		IF bPackBarcode THEN
			sOutBarcode	:= sPackBarcode;
		ELSIF bOuterBarcode THEN
			sOutBarcode := F_CODE_GetItem(sOuterBarcode, eCodeAIType.SerialCode, stCodeInfo_Outer);
		ELSIF bCaseBarcode THEN
			(*fbDecodeGS1(strGS1String := CONCAT(']d2',sCaseBarcode), bDontParseAsGS1 := TRUE, strBarcode => sOutBarcode);*)
			sOutBarcode	:= sCaseBarcode;
		ELSE
			sOutBarcode := '';
		END_IF

		bScanDone := TRUE;

	ELSIF bEnableInvalidSearch AND NOT bEnableCaseContentSearch AND NOT bEnablePackCodeRefeed THEN

		sNewPackCodeRefeed := '';

		IF bPackBarcode THEN
			sOutBarcode :=  F_CODE_GetItem(sPackBarcode, eCodeAIType.SerialCode, stCodeInfo_Pack);
		ELSIF bOuterIntermediate THEN
			sOutBarcode := F_CODE_GetItem(sOuterIntermediateBarcode, eCodeAIType.SerialCode, stCodeInfo_Intermediate);
		ELSIF bOuterBarcode THEN
			sOutBarcode := F_CODE_GetItem(sOuterBarcode, eCodeAIType.SerialCode, stCodeInfo_Outer);
		ELSE
			sOutBarcode := '';
		END_IF

		bScanDone := TRUE;

	ELSIF bEnableInvalidSearch AND NOT bEnableCaseContentSearch AND bEnablePackCodeRefeed THEN

		IF bPackBarcode THEN
			sOutBarcode := F_CODE_GetItem(sPackBarcode, eCodeAIType.SerialCode, stCodeInfo_Pack);
			sNewPackCodeRefeed := sPackBarcode;
		ELSE
			sOutBarcode := '';
			sNewPackCodeRefeed := '';
		END_IF

		bScanDone := TRUE;

	ELSE

		sOutBarcode := '';
		sNewPackCodeRefeed := '';

	END_IF

	(* set output *)
	bBusy := FALSE;
	bDone := TRUE;
END_IF

END_FUNCTION_BLOCK

// ---- POUs/METS/Common LIB/09_SYSTEM LIB/FB_SYSTEM_SeqControl.TcPOU
FUNCTION_BLOCK FB_SYSTEM_SeqControl
VAR_INPUT
	nSeqStepNo	: INT;
END_VAR
VAR_OUTPUT
	bActive		: BOOL;
	bStep00		: BOOL;
	bStep01		: BOOL;
	bStep02		: BOOL;
	bStep03		: BOOL;
	bStep04		: BOOL;
	bStep05		: BOOL;
	bStep06		: BOOL;
	bStep07		: BOOL;
	bStep08		: BOOL;
	bStep09		: BOOL;
	bStep10		: BOOL;
	bStep11		: BOOL;
	bStep12		: BOOL;
	bStep13		: BOOL;
	bStep14		: BOOL;
	bStep15		: BOOL;
	bStep16		: BOOL;
	bStep17		: BOOL;
	bStep18		: BOOL;
	bStep19		: BOOL;
	bStep20		: BOOL;
END_VAR
VAR
END_VAR
(*
-------------------------------------------------------------------------------------------------
Date		Version	Author	Comments
-------------------------------------------------------------------------------------------------
30/01/2015	3.00.00	PB		Initial release

-------------------------------------------------------------------------------------------------
*)

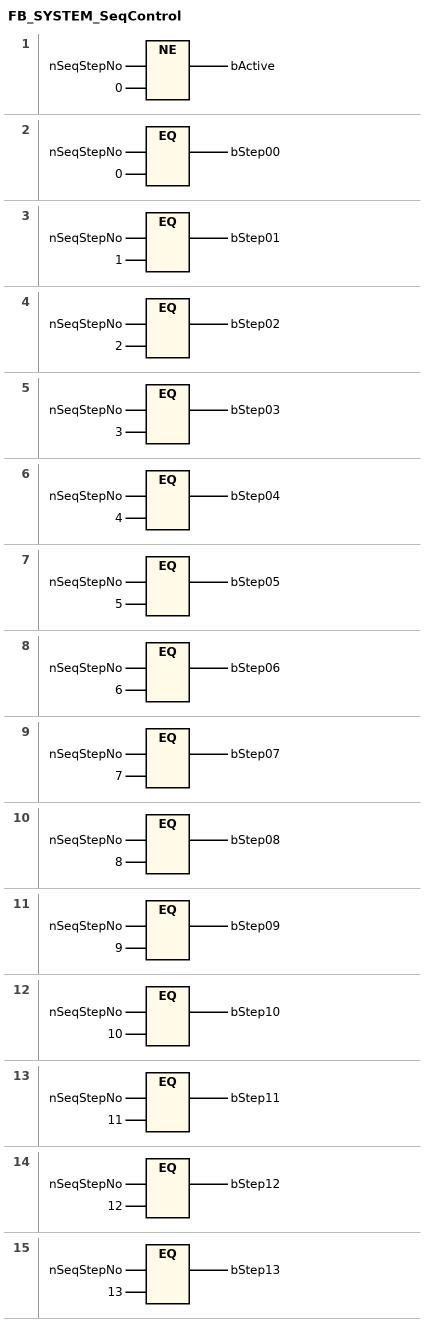
// NETWORK 1
bActive := nSeqStepNo <> 0;

// NETWORK 2
bStep00 := nSeqStepNo = 0;

// NETWORK 3
bStep01 := nSeqStepNo = 1;

// NETWORK 4
bStep02 := nSeqStepNo = 2;

// NETWORK 5
bStep03 := nSeqStepNo = 3;

// NETWORK 6
bStep04 := nSeqStepNo = 4;

// NETWORK 7
bStep05 := nSeqStepNo = 5;

// NETWORK 8
bStep06 := nSeqStepNo = 6;

// NETWORK 9
bStep07 := nSeqStepNo = 7;

// NETWORK 10
bStep08 := nSeqStepNo = 8;

// NETWORK 11
bStep09 := nSeqStepNo = 9;

// NETWORK 12
bStep10 := nSeqStepNo = 10;

// NETWORK 13
bStep11 := nSeqStepNo = 11;

// NETWORK 14
bStep12 := nSeqStepNo = 12;

// NETWORK 15
bStep13 := nSeqStepNo = 13;

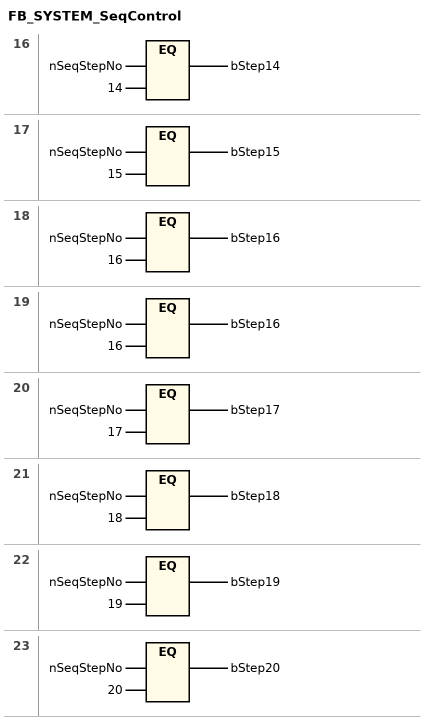
// NETWORK 16
bStep14 := nSeqStepNo = 14;

// NETWORK 17
bStep15 := nSeqStepNo = 15;

// NETWORK 18
bStep16 := nSeqStepNo = 16;

// NETWORK 19
bStep16 := nSeqStepNo = 16;

// NETWORK 20
bStep17 := nSeqStepNo = 17;

// NETWORK 21
bStep18 := nSeqStepNo = 18;

// NETWORK 22
bStep19 := nSeqStepNo = 19;

// NETWORK 23
bStep20 := nSeqStepNo = 20;

END_FUNCTION_BLOCK

// ---- POUs/METS/Common LIB/09_SYSTEM LIB/FB_SYSTEM_ShiftMonitor.TcPOU
FUNCTION_BLOCK FB_SYSTEM_ShiftMonitor
VAR_INPUT
	bEnable				: BOOL;
	stSystemTime			: TIMESTRUCT;
END_VAR
VAR_IN_OUT

	stPCMStatus				: ST_PCM_Status;	(* PCMstatus *)
	aShiftSchedule				: ARRAY[1..cSHIFTNUMBER] OF TIMESTRUCT;
	aShiftChangeActive		: ARRAY[1..cSHIFTNUMBER] OF BOOL;
	stCurrentStatisticNV		: ST_NOVRAM_METS_EventCounters;
	stCSVStoreTable			: ST_HMI_CSVStoreTable;

END_VAR
VAR_OUTPUT

	bShiftChanged				: BOOL;
	stLastShift					: TIMESTRUCT;
END_VAR
VAR
	fbExecute					: R_TRIG;
	nNumberShift				: T_PositiveINT;
	bEndOfShift				: BOOL;
	(*nActiveShiftCounter		: INT;*)

END_VAR

(* shift manager disabled *)
IF NOT bEnable  THEN

	(* clear outputs *)
	bEndOfShift := FALSE;
	MEMSET(ADR(stLastShift), 16#00, SIZEOF(stLastShift));
	RETURN;
END_IF


IF stCurrentStatisticNV.stEventStartDT.wYear = 0 AND stCurrentStatisticNV.stEventStartDT.wMonth = 0 THEN
	stCurrentStatisticNV.stEventStartDT := stSystemTime;
	stCurrentStatisticNV.nShiftID 		:= 1;
END_IF
(*
nActiveShiftCounter := 0;

FOR nNumberShift := 1 TO cSHIFTNUMBER DO

	IF	aShiftChangeActive[nNumberShift] 	THEN
		nActiveShiftCounter := nActiveShiftCounter + 1;
	END_IF
END_FOR
*)
FOR nNumberShift := 1 TO cSHIFTNUMBER DO

	IF	aShiftChangeActive[nNumberShift] 							AND
		aShiftSchedule[nNumberShift].wHour  = stSystemTime.wHour 		AND
		aShiftSchedule[nNumberShift].wMinute = stSystemTime.wMinute 	(*AND
		aShiftSchedule[nNumberShift].wSecond = .sSystemTime.wSecond*)		THEN

		(*stCurrentStatisticNV.stEventEndDT	:= stSystemTime;*)
		bEndOfShift := TRUE;
		EXIT;
	ELSE
		bEndOfShift := FALSE;
	END_IF
END_FOR

(*
IF nActiveShiftCounter <> 0 THEN
	stCurrentStatisticNV.stEndShiftDT := F_ApplyTimeOffset(stCurrentStatisticNV.stStartShiftDT, 86400000/nActiveShiftCounter);
ELSE
	stCurrentStatisticNV.stEndShiftDT := F_ApplyTimeOffset(stCurrentStatisticNV.stStartShiftDT, 86400000);
END_IF
*)
(***************************Store current data to CSV structure for HMI******************************************)
fbExecute(CLK := bEndOfShift );

(* rising edge detected *)
IF fbExecute.Q = TRUE THEN

(*Blok przepisywania danych do  struct*)
	stCSVStoreTable.nShiftID 	:= 	stCurrentStatisticNV.nShiftID;
	stCSVStoreTable.sRSKU	:=	stCurrentStatisticNV.sRSKU;
	stCSVStoreTable.sProductionOrder	:=	stCurrentStatisticNV.sProductionOrder;

	stCSVStoreTable.stEventStartDT 	:= stCurrentStatisticNV.stEventStartDT;
	stCSVStoreTable.stEventEndDT 	:= stSystemTime;

	MEMCPY(ADR(stCSVStoreTable.stMachineStateStatistic), ADR(stCurrentStatisticNV.stMachineStateStatistic), SIZEOF(stCSVStoreTable.stMachineStateStatistic));
	MEMCPY(ADR(stCSVStoreTable.aGeneralKPIStatistic), ADR(stCurrentStatisticNV.aGeneralKPIStatistic), SIZEOF(stCSVStoreTable.aGeneralKPIStatistic));
	MEMCPY(ADR(stCSVStoreTable.aAlarmsStatistic), ADR(stCurrentStatisticNV.aAlarmsStatistic), SIZEOF(stCSVStoreTable.aAlarmsStatistic));
	MEMCPY(ADR(stCSVStoreTable.aRejectCounters), ADR(stCurrentStatisticNV.aRejectCounters), SIZEOF(stCSVStoreTable.aRejectCounters));

	stCSVStoreTable.bDataStoredByHMI := TRUE;

	stLastShift	:= stCSVStoreTable.stEventEndDT ;
	MEMSET(ADR(stCurrentStatisticNV), 16#00, SIZEOF(stCurrentStatisticNV));

	stCurrentStatisticNV.nShiftID 				:= nNumberShift;
	stCurrentStatisticNV.sRSKU 				:= stPCMStatus.sRetailSKU;
	stCurrentStatisticNV.sProductionOrder  	:= stPCMStatus.sProductionOrder;

	stCurrentStatisticNV.stEventStartDT 		:= stSystemTime;

	bShiftChanged	:=TRUE;
ELSE
	bShiftChanged	:=FALSE;
END_IF

END_FUNCTION_BLOCK

// ---- POUs/METS/Common LIB/09_SYSTEM LIB/FB_SYSTEM_ValidateSettings.TcPOU
(* loads XML settings file and validates data *)
FUNCTION_BLOCK FB_SYSTEM_ValidateSettings
VAR_INPUT
	bExecute				: BOOL;			(* set TRUE to read XML file into Settings *)
	//strBasePath			: STRING(255);
END_VAR
VAR_IN_OUT
	stMetsStatus			: ST_SYSTEM_MachineStatus;	(* settings data structure *)
	stMachineConfig		: ST_SYSTEM_Config;
	stMachineDevices		: ST_SYSTEM_DeviceState;
END_VAR
VAR_OUTPUT
	bDone				: BOOL;			(* TRUE = load product instruction complete *)
	bError				: BOOL;			(* TRUE = error with process *)
	bValid				: BOOL;			(* TRUE = settings validated OK, not reset when bExecute goes FALSE *)
	strFieldName			: STRING(20);		(* field where validation error occurred, not reset when bExecute goes FALSE *)
	strFieldData			: STRING(20);		(* data that failed validation, not reset when bExecute goes FALSE *)
END_VAR
VAR
	fbExecute				: R_TRIG;
	nIndex				: INT;
	nCharPos				: INT;
END_VAR

fbExecute(CLK := bExecute);
IF fbExecute.Q = TRUE THEN

	(* clear outputs *)
	bDone := FALSE;
	bError := FALSE;

(* <ProductionLine><PCM> field contains data *)
	IF LEN(stMachineConfig.stProductionLine.sPCM) > 0 THEN

		(* set PCM enabled and generate PCM base path, current PCM file name and new PCM file name template*)
		stMetsStatus.stPCMStatus.bEnabled := TRUE;
		stMetsStatus.stPCMStatus.sPCMCurrent := F_CONCAT5('PCM_', stMachineConfig.sProductionSite, '_', stMachineConfig.stProductionLine.sPCM, '_Current.xml');
		stMetsStatus.stPCMStatus.sPCMTemplate := F_CONCAT5('PCM_', stMachineConfig.sProductionSite, '_', stMachineConfig.stProductionLine.sPCM, '_????????_??????.xml');

	(* <ProductionLine><OPI> field is blank *)
	ELSE
		bError := TRUE;
		(* clear OPIStatus and OPI *)
		MEMSET(ADR(stMetsStatus.stPCMStatus), 16#00, SIZEOF(stMetsStatus.stPCMStatus));
		MEMSET(ADR(stMetsStatus.stPCMData), 16#00, SIZEOF(stMetsStatus.stPCMData));
	END_IF

(* sShiftOffsetTime contains data *)
	IF LEN(stMachineConfig.sShiftOffsetTime) > 0 THEN

		(* sShiftOffsetTime must be in format of '+hh:mm' or '-hh:mm' *)
		nCharPos := FIND(stMachineConfig.sShiftOffsetTime, ':');

		(* ':' char found *)
		IF nCharPos > 1 THEN
			IF  STRING_TO_DINT(LEFT(stMachineConfig.sShiftOffsetTime, nCharPos - 1)) > -12
				AND STRING_TO_DINT(LEFT(stMachineConfig.sShiftOffsetTime, nCharPos - 1)) < 12
				AND STRING_TO_DINT(RIGHT(stMachineConfig.sShiftOffsetTime, LEN(stMachineConfig.sShiftOffsetTime) - nCharPos)) < 12THEN

				(* convert sShiftOffsetTime to DINT where 1000 = 1s *)
				stMetsStatus.nShiftOffsetTime := (STRING_TO_DINT(LEFT(stMachineConfig.sShiftOffsetTime, nCharPos - 1)) * 3600000) +
												(STRING_TO_DINT(RIGHT(stMachineConfig.sShiftOffsetTime, LEN(stMachineConfig.sShiftOffsetTime) - nCharPos)) * 60000);
			ELSE
				(* reset to 0 with correct format *)
				stMachineConfig.sShiftOffsetTime := '+00:00';
				stMetsStatus.nShiftOffsetTime := 0;
			END_IF
				(*nCharPos := FIND(stMachineConfig.sShiftOffsetTime, '-');
				IF nCharPos > 0 THEN
					stMetsStatus.nShiftOffsetTime := stMetsStatus.nShiftOffsetTime *-1;
				END_IF*)
		(* incorrect format *)
		ELSE
			(* reset to 0 with correct format *)
			stMachineConfig.sShiftOffsetTime := '+00:00';
			stMetsStatus.nShiftOffsetTime := 0;
		END_IF
	(* sShiftOffsetTime is empty *)
	ELSE
		(* eet to 0 with correct format *)
		stMachineConfig.sShiftOffsetTime := '+00:00';
		stMetsStatus.nShiftOffsetTime := 0;
	END_IF

(* check if Case advance settings are in proper range*)
	stMachineConfig.nCaseQueueLength := LIMIT(1, stMachineConfig.nCaseQueueLength, cMAX_CASE_QUEUE);
	stMachineConfig.nCaseContentBuffer := LIMIT(0, stMachineConfig.nCaseContentBuffer, 4);

	(* settings validated OK *)
	IF bError = FALSE THEN

		(* status outputs *)
		bValid:= TRUE;
		strFieldData := 'Settings OK';
		strFieldName:= 'Settings OK';

		(* determine which cameras are configured *)
		FOR nIndex := 1 TO cMAX_CAMERA_NUMBER DO

			(* check if Scanner2D device is configured *)
			stMachineDevices.aCameraIPSettingsValid[nIndex] := F_IP_AddressPort(stMachineConfig.aCameraSettings[nIndex].stCameraIP.IP, stMachineConfig.aCameraSettings[nIndex].stCameraIP.Port);

		END_FOR

		FOR nIndex := 1 TO cMAX_HAND_SCANNERS  DO

			(* check if HandScanner device is configured *)
			stMachineDevices.aHandScannersValid[nIndex] := stMachineConfig.aHandScannersConfig[1].nBaudRate <> 0;

		END_FOR

		FOR nIndex := 1 TO cMAX_PRINTER_NUMBER DO

			(* check if Printer device is configured *)
			stMachineDevices.aPrinterIPSettingsValid[nIndex] := F_IP_AddressPort(stMachineConfig.aPrinterSettings[nIndex].stIPAdressPort.IP, stMachineConfig.aPrinterSettings[nIndex].stIPAdressPort.Port);

		END_FOR

	(* Settings are invalid *)
	ELSE

		(* status output *)
		bValid := FALSE;
		strFieldData := 'Settings Not Valide';
		strFieldName:= 'Settings Not Valide';

		(* clear devices configured array *)
		MEMSET(ADR(stMachineDevices), 16#00, SIZEOF(stMachineDevices));
	END_IF

	bDone := TRUE;

(* bExecute has been reset *)
ELSIF bExecute = FALSE THEN

	bDone := FALSE;
	bError := FALSE;
END_IF

END_FUNCTION_BLOCK

// ---- POUs/_Exclude/C09_MaintainFolders_OLD.TcPOU
(* delete old files and delete oldest files if number of files exceeds specified number *)
PROGRAM C09_MaintainFolders_OLD
VAR
	tArchiveCheck				: TIME := t#4s;
	fbMaintainArchive			: FB_PulseGenerator;
	tDeleteTimeCheck			: TIME := t#20m;
	fbMaintainDeleteTime		: FB_PulseGenerator;
	(*tDeleteItemCheck			: TIME := t#4s;
	fbMaintainDeleteItem		: FB_PulseGenerator;*)
	nActivateBitWord			: DWORD; (* if index increase 32 bits it is necceasry to declar 64 bits var like LREAL;*)

	aMaintainFolders			: ARRAY[1..17] OF NT_StartProcess;
	aManualMaintain			: ARRAY[1..17] OF BOOL;
	(*fbMoveOHMToArchive		: FB_OHM_MoveToArchive;*)
	(*fbMoveCACToArchive		: FB_CAC_MoveToArchive;*)
	fbMoveCHMToArchive		: FB_CHM_MoveToArchive;
	bZipCHMArchive			: BOOL;
	rtrigZipAfetrPassthrough		: R_TRIG;
	bManualZip					: BOOL;

	(*fbCompresOHMArchive		: NT_StartProcess;
	fbCompresCHMArchive		: NT_StartProcess;
	fbCompresPHMArchive		: NT_StartProcess;

	fbDeleteCHMNoLabel		: NT_StartProcess;*)

	fbRestoreTimer			: TON;
	fbRestoreOACFromCAC		: FB_CAC_RestoreOAC;
	nOCVFilesRestored			: UDINT;
	nOACFilesRestored			: UDINT;
	nCACFilesRestored			: UDINT;

	(*rtrigClearOCV				: R_TRIG;
	rtrigClearOCVError			: R_TRIG;
	rtrigClearOAC				: R_TRIG;
	rtrigClearOACError			: R_TRIG;

	fbClearOCVArchive			: FB_OCV_ClearArchive;
	fbClearOCVError			: FB_OCV_ClearArchive;
	fbClearOACArchive			: FB_OAC_ClearArchive;
	fbClearOACError			: FB_OAC_ClearArchive;

	rtrigClearOHM_FLG			: R_TRIG;
	rtrigClearCHM_FLG			: R_TRIG;

	fbClearOHM_FLG			: FB_OHM_ClearFLG;
	fbClearCHM_FLG			: FB_CHM_ClearFLG;
	btest : BOOL;*)

(********************************************************************************
		cBASE_FOLDER_ARR	: ARRAY[1..cSYSTEM_FOLDER_LIMIT] OF T_FolderName :=
			(*01*)'Bridge\',		(*02*)'Bridge\Archive\',		(*03*)'Bridge\Restore\',
			(*04*)'CAC\',		(*05*)'CAC\Archive\',		(*06*)'CAC\Error\',		(*07*)'CAC\Restore\', 	(*08*)'CAC\Restore\Archive\',
			(*09*)'CHM\',		(*10*)'CHM\Archive\',		(*11*)'CHM\Error\',		(*12*)'CHM\OK\',		(*13*)'CHM\Commissioning_Mode\',
			(*14*)'HMI\',
			(*15*)'KPI\',		(*16*)'KPI\Archive\',			(*17*)'KPI\Shift\',		(*18*)'KPI\ProdOrder\',
			(*19*)'OAC\',		(*20*)'OAC\Error\',
			(*21*)'OCV\',		(*22*)'OCV\Error\',
			(*23*)'OHM\',		(*24*)'OHM\Archive\',		(*25*)'OHM\Error\',		(*26*)'OHM\OK\',		(*27*)'OHM\Pending\',
			(*28*)'PCM\',		(*29*)'PCM\Archive\',		(*30*)'PCM\Error\',		(*31*)'PCM\Incoming\',
			(*32*)'PAC\',
			(*33*)'PHM\',		(*34*)'PHM\Archive\',		(*35*)'PHM\Error\',		(*36*)'PHM\OK\',
			(*37*)'Settings\',	(*38*)'Settings\Backups\',
			(*39*)'Templates\',
			(*40*)'Orca\',
			(*41*) 'SystemLog\';

*************************************************************************************)
(********************************************************************************
Delete Items
	DeleteItem <path> <filesToKeep> [createLog] [deleteDirs] [dirsToKeep]
	path: Directory path
	filesToKeep: Number OF files TO RETAIN
	createLog: (Optional) Boolean to enable logging
	deleteDirs: (Optional) Boolean to include directories
	dirsToKeep: (Optional) Number of directories to retain

Delete by Time
	DeleteTime <path> <fileAge> [createLog] [deleteDirs] [ageUnit]
	path: Directory path
	fileAge: Maximum age of files to retain
	createLog: (Optional) Boolean to enable logging
	deleteDirs: (Optional) Boolean to include inside directories for file search
	ageUnit: (Optional) Time unit for age values (Day/Hour/Minute), defaults to Day

Archive
	Archive <chmArchiveFolder> <lastArchiveDateName> [createLog]
	chmArchiveFolder: Archive folder path
	lastArchiveDateName: Last archive date identifier
	createLog: (Optional) Boolean TO enable logging
*************************************************************************************)
END_VAR

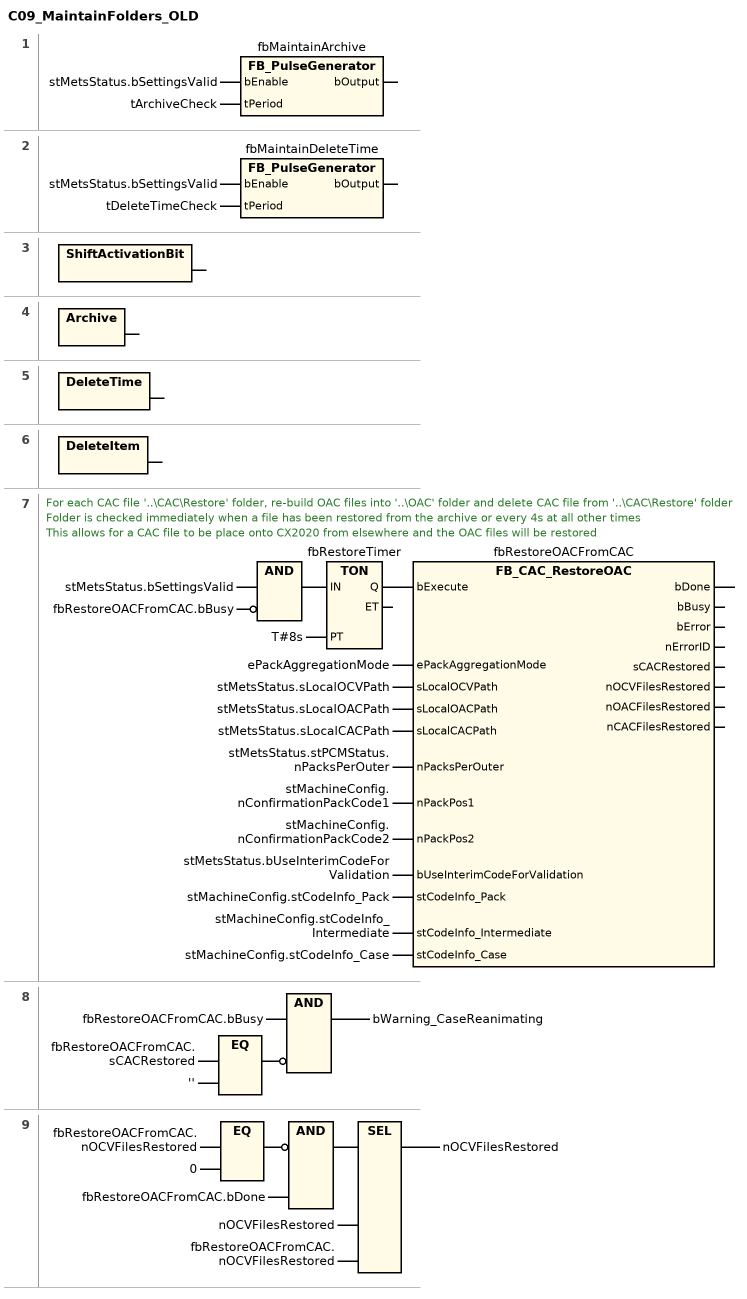
// NETWORK 1
fbMaintainArchive(bEnable := stMetsStatus.bSettingsValid, tPeriod := tArchiveCheck); // FB_PulseGenerator

// NETWORK 2
fbMaintainDeleteTime(bEnable := stMetsStatus.bSettingsValid, tPeriod := tDeleteTimeCheck); // FB_PulseGenerator

// NETWORK 3
ShiftActivationBit();

// NETWORK 4
Archive();

// NETWORK 5
DeleteTime();

// NETWORK 6
DeleteItem();

// NETWORK 7
// 					For each CAC file '..\CAC\Restore' folder, re-build OAC files into '..\OAC' folder and delete CAC file from '..\CAC\Restore' folder
// Folder is checked immediately when a file has been restored from the archive or every 4s at all other times
// This allows for a CAC file to be place onto CX2020 from elsewhere and the OAC files will be restored
//
fbRestoreTimer(IN := stMetsStatus.bSettingsValid AND NOT fbRestoreOACFromCAC.bBusy, PT := T#8s); // TON
fbRestoreOACFromCAC(
    bExecute := fbRestoreTimer.Q,
    ePackAggregationMode := ePackAggregationMode,
    sLocalOCVPath := stMetsStatus.sLocalOCVPath,
    sLocalOACPath := stMetsStatus.sLocalOACPath,
    sLocalCACPath := stMetsStatus.sLocalCACPath,
    nPacksPerOuter := stMetsStatus.stPCMStatus.nPacksPerOuter,
    nPackPos1 := stMachineConfig.nConfirmationPackCode1,
    nPackPos2 := stMachineConfig.nConfirmationPackCode2,
    bUseInterimCodeForValidation := stMetsStatus.bUseInterimCodeForValidation,
    stCodeInfo_Pack := stMachineConfig.stCodeInfo_Pack,
    stCodeInfo_Intermediate := stMachineConfig.stCodeInfo_Intermediate,
    stCodeInfo_Case := stMachineConfig.stCodeInfo_Case); // FB_CAC_RestoreOAC

// NETWORK 8
bWarning_CaseReanimating := fbRestoreOACFromCAC.bBusy AND NOT (fbRestoreOACFromCAC.sCACRestored = '');

// NETWORK 9
nOCVFilesRestored := SEL(NOT (fbRestoreOACFromCAC.nOCVFilesRestored = 0) AND fbRestoreOACFromCAC.bDone, nOCVFilesRestored, fbRestoreOACFromCAC.nOCVFilesRestored);

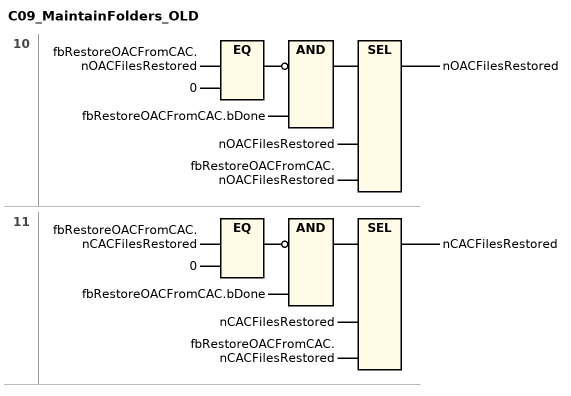
// NETWORK 10
nOACFilesRestored := SEL(NOT (fbRestoreOACFromCAC.nOACFilesRestored = 0) AND fbRestoreOACFromCAC.bDone, nOACFilesRestored, fbRestoreOACFromCAC.nOACFilesRestored);

// NETWORK 11
nCACFilesRestored := SEL(NOT (fbRestoreOACFromCAC.nCACFilesRestored = 0) AND fbRestoreOACFromCAC.bDone, nCACFilesRestored, fbRestoreOACFromCAC.nCACFilesRestored);

ACTION Archive:
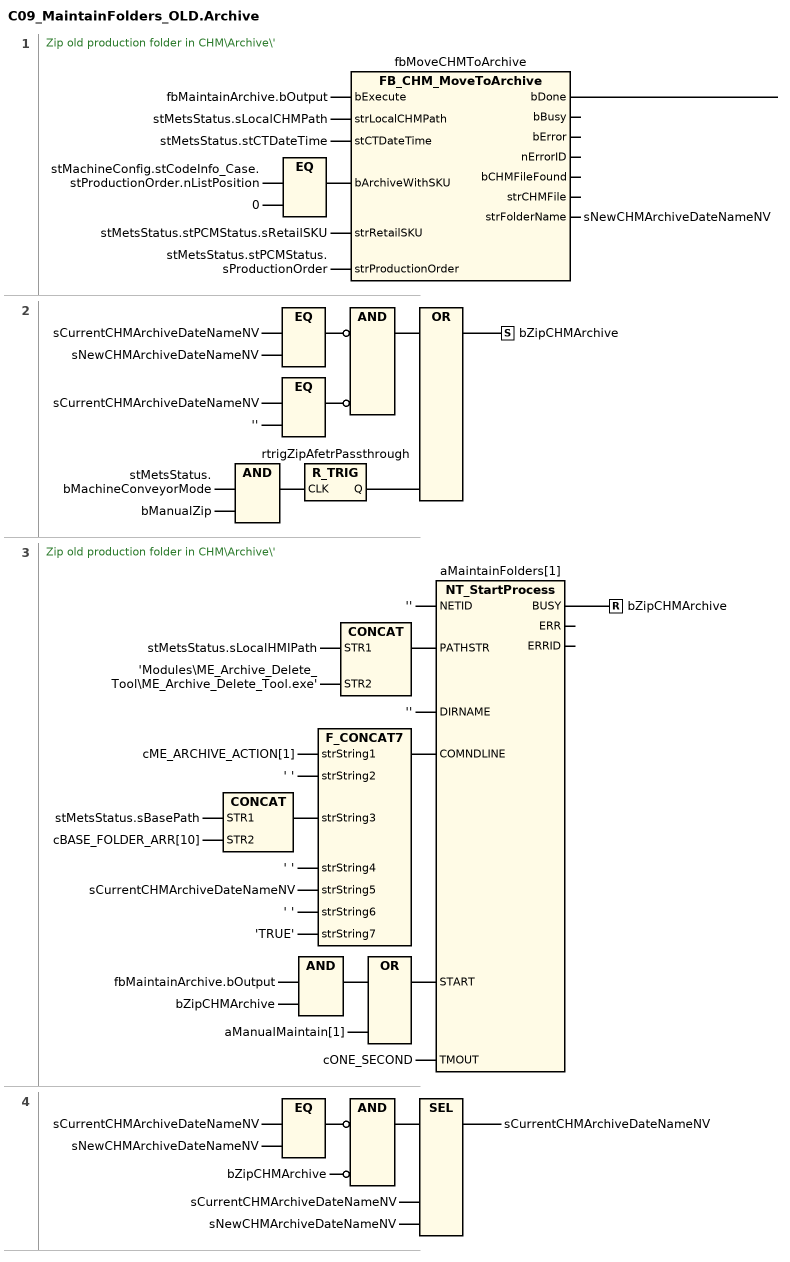
// NETWORK 1
// 					Zip old production folder in CHM\Archive\'
//
//
fbMoveCHMToArchive(
    bExecute := fbMaintainArchive.bOutput,
    strLocalCHMPath := stMetsStatus.sLocalCHMPath,
    stCTDateTime := stMetsStatus.stCTDateTime,
    bArchiveWithSKU := stMachineConfig.stCodeInfo_Case.stProductionOrder.nListPosition = 0,
    strRetailSKU := stMetsStatus.stPCMStatus.sRetailSKU,
    strProductionOrder := stMetsStatus.stPCMStatus.sProductionOrder,
    strFolderName => sNewCHMArchiveDateNameNV); // FB_CHM_MoveToArchive

// NETWORK 2
rtrigZipAfetrPassthrough(CLK := stMetsStatus.bMachineConveyorMode AND bManualZip); // R_TRIG
bZipCHMArchive S= NOT (sCurrentCHMArchiveDateNameNV = sNewCHMArchiveDateNameNV) AND NOT (sCurrentCHMArchiveDateNameNV = '') OR rtrigZipAfetrPassthrough.Q;

// NETWORK 3
// Zip old production folder in CHM\Archive\'
aMaintainFolders[1](
    NETID := '',
    PATHSTR := CONCAT(STR1 := stMetsStatus.sLocalHMIPath, STR2 := 'Modules\ME_Archive_Delete_Tool\ME_Archive_Delete_Tool.exe'),
    DIRNAME := '',
    COMNDLINE := F_CONCAT7(strString1 := cME_ARCHIVE_ACTION[1], strString2 := ' ', strString3 := CONCAT(STR1 := stMetsStatus.sBasePath, STR2 := cBASE_FOLDER_ARR[10]), strString4 := ' ', strString5 := sCurrentCHMArchiveDateNameNV, strString6 := ' ', strString7 := 'TRUE'),
    START := fbMaintainArchive.bOutput AND bZipCHMArchive OR aManualMaintain[1],
    TMOUT := cONE_SECOND); // NT_StartProcess
bZipCHMArchive R= aMaintainFolders[1].BUSY;

// NETWORK 4
sCurrentCHMArchiveDateNameNV := SEL(NOT (sCurrentCHMArchiveDateNameNV = sNewCHMArchiveDateNameNV) AND NOT bZipCHMArchive, sCurrentCHMArchiveDateNameNV, sNewCHMArchiveDateNameNV);
END_ACTION

ACTION DeleteItem:
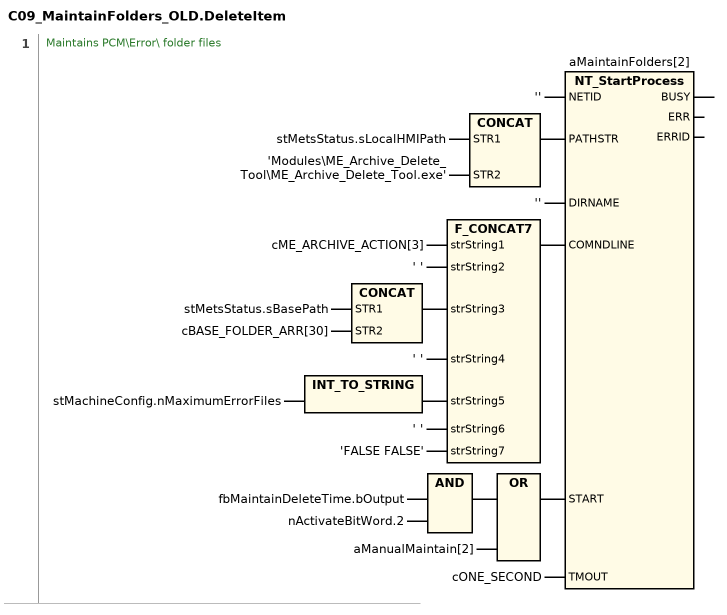
// NETWORK 1
// Maintains PCM\Error\ folder files
aMaintainFolders[2](
    NETID := '',
    PATHSTR := CONCAT(STR1 := stMetsStatus.sLocalHMIPath, STR2 := 'Modules\ME_Archive_Delete_Tool\ME_Archive_Delete_Tool.exe'),
    DIRNAME := '',
    COMNDLINE := F_CONCAT7(strString1 := cME_ARCHIVE_ACTION[3], strString2 := ' ', strString3 := CONCAT(STR1 := stMetsStatus.sBasePath, STR2 := cBASE_FOLDER_ARR[30]), strString4 := ' ', strString5 := INT_TO_STRING(stMachineConfig.nMaximumErrorFiles), strString6 := ' ', strString7 := 'FALSE FALSE'),
    START := fbMaintainDeleteTime.bOutput AND nActivateBitWord.2 OR aManualMaintain[2],
    TMOUT := cONE_SECOND); // NT_StartProcess

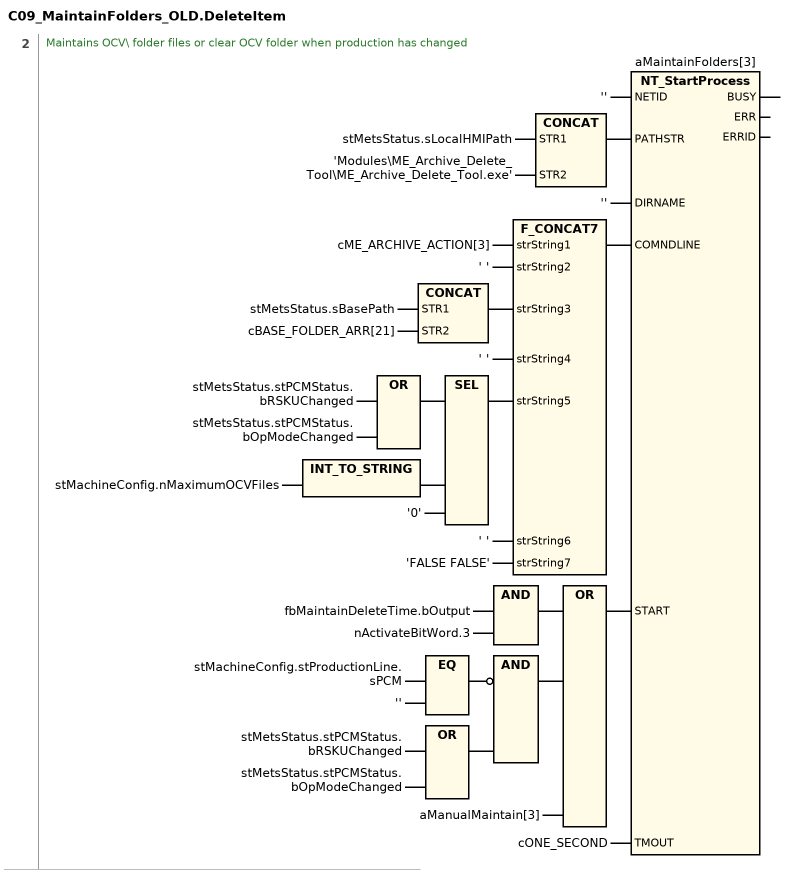
// NETWORK 2
// Maintains OCV\ folder files or clear OCV folder when production has changed
aMaintainFolders[3](
    NETID := '',
    PATHSTR := CONCAT(STR1 := stMetsStatus.sLocalHMIPath, STR2 := 'Modules\ME_Archive_Delete_Tool\ME_Archive_Delete_Tool.exe'),
    DIRNAME := '',
    COMNDLINE := F_CONCAT7(strString1 := cME_ARCHIVE_ACTION[3], strString2 := ' ', strString3 := CONCAT(STR1 := stMetsStatus.sBasePath, STR2 := cBASE_FOLDER_ARR[21]), strString4 := ' ', strString5 := SEL(stMetsStatus.stPCMStatus.bRSKUChanged OR stMetsStatus.stPCMStatus.bOpModeChanged, INT_TO_STRING(stMachineConfig.nMaximumOCVFiles), '0'), strString6 := ' ', strString7 := 'FALSE FALSE'),
    START := fbMaintainDeleteTime.bOutput AND nActivateBitWord.3 OR NOT (stMachineConfig.stProductionLine.sPCM = '') AND (stMetsStatus.stPCMStatus.bRSKUChanged OR stMetsStatus.stPCMStatus.bOpModeChanged) OR aManualMaintain[3],
    TMOUT := cONE_SECOND); // NT_StartProcess

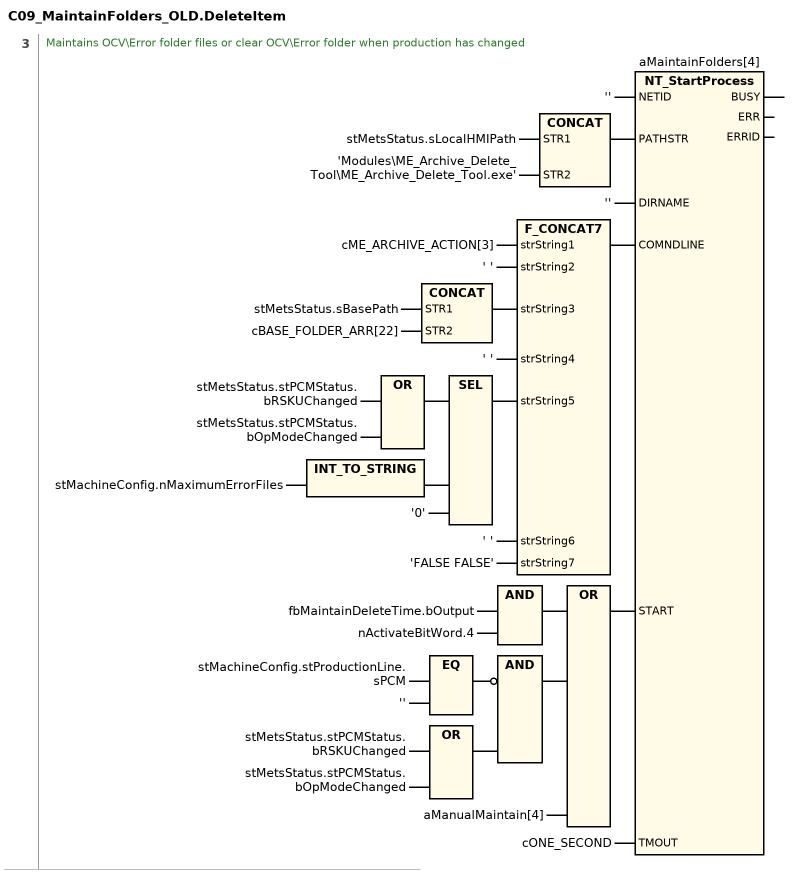
// NETWORK 3
// Maintains OCV\Error folder files or clear OCV\Error folder when production has changed
aMaintainFolders[4](
    NETID := '',
    PATHSTR := CONCAT(STR1 := stMetsStatus.sLocalHMIPath, STR2 := 'Modules\ME_Archive_Delete_Tool\ME_Archive_Delete_Tool.exe'),
    DIRNAME := '',
    COMNDLINE := F_CONCAT7(strString1 := cME_ARCHIVE_ACTION[3], strString2 := ' ', strString3 := CONCAT(STR1 := stMetsStatus.sBasePath, STR2 := cBASE_FOLDER_ARR[22]), strString4 := ' ', strString5 := SEL(stMetsStatus.stPCMStatus.bRSKUChanged OR stMetsStatus.stPCMStatus.bOpModeChanged, INT_TO_STRING(stMachineConfig.nMaximumErrorFiles), '0'), strString6 := ' ', strString7 := 'FALSE FALSE'),
    START := fbMaintainDeleteTime.bOutput AND nActivateBitWord.4 OR NOT (stMachineConfig.stProductionLine.sPCM = '') AND (stMetsStatus.stPCMStatus.bRSKUChanged OR stMetsStatus.stPCMStatus.bOpModeChanged) OR aManualMaintain[4],
    TMOUT := cONE_SECOND); // NT_StartProcess

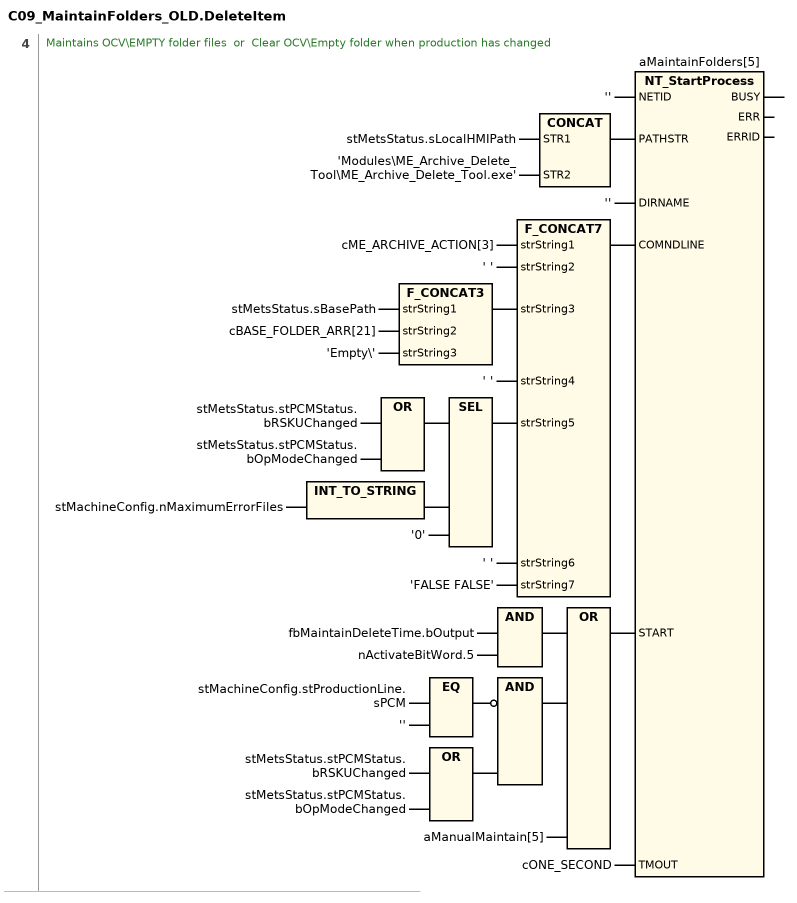
// NETWORK 4
// Maintains OCV\EMPTY folder files  or  Clear OCV\Empty folder when production has changed
aMaintainFolders[5](
    NETID := '',
    PATHSTR := CONCAT(STR1 := stMetsStatus.sLocalHMIPath, STR2 := 'Modules\ME_Archive_Delete_Tool\ME_Archive_Delete_Tool.exe'),
    DIRNAME := '',
    COMNDLINE := F_CONCAT7(strString1 := cME_ARCHIVE_ACTION[3], strString2 := ' ', strString3 := F_CONCAT3(strString1 := stMetsStatus.sBasePath, strString2 := cBASE_FOLDER_ARR[21], strString3 := 'Empty\'), strString4 := ' ', strString5 := SEL(stMetsStatus.stPCMStatus.bRSKUChanged OR stMetsStatus.stPCMStatus.bOpModeChanged, INT_TO_STRING(stMachineConfig.nMaximumErrorFiles), '0'), strString6 := ' ', strString7 := 'FALSE FALSE'),
    START := fbMaintainDeleteTime.bOutput AND nActivateBitWord.5 OR NOT (stMachineConfig.stProductionLine.sPCM = '') AND (stMetsStatus.stPCMStatus.bRSKUChanged OR stMetsStatus.stPCMStatus.bOpModeChanged) OR aManualMaintain[5],
    TMOUT := cONE_SECOND); // NT_StartProcess

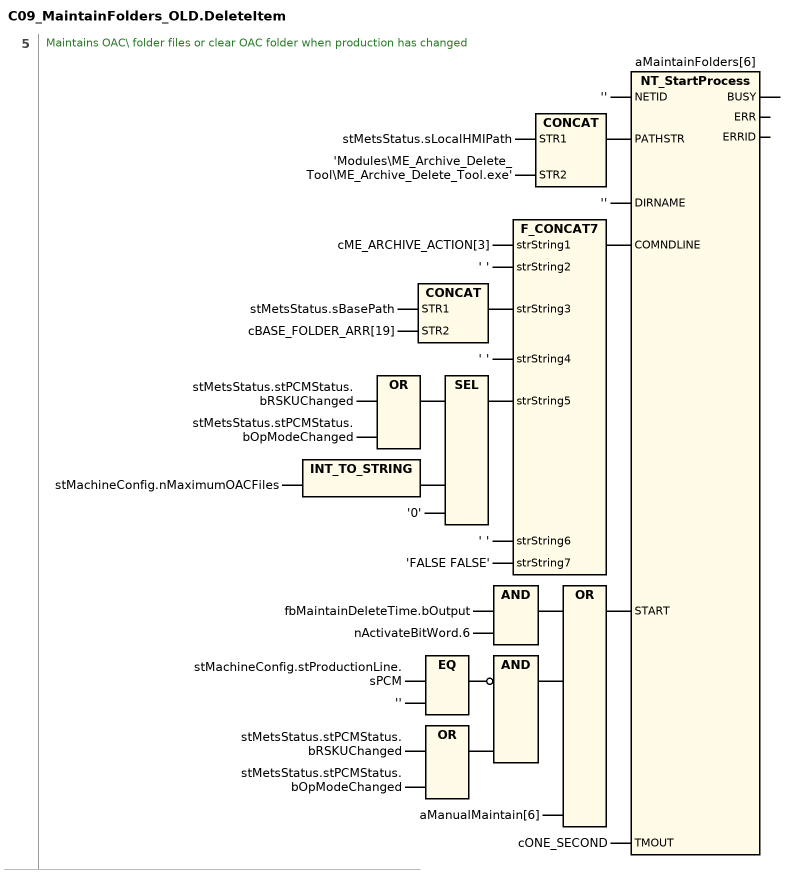
// NETWORK 5
// Maintains OAC\ folder files or clear OAC folder when production has changed
aMaintainFolders[6](
    NETID := '',
    PATHSTR := CONCAT(STR1 := stMetsStatus.sLocalHMIPath, STR2 := 'Modules\ME_Archive_Delete_Tool\ME_Archive_Delete_Tool.exe'),
    DIRNAME := '',
    COMNDLINE := F_CONCAT7(strString1 := cME_ARCHIVE_ACTION[3], strString2 := ' ', strString3 := CONCAT(STR1 := stMetsStatus.sBasePath, STR2 := cBASE_FOLDER_ARR[19]), strString4 := ' ', strString5 := SEL(stMetsStatus.stPCMStatus.bRSKUChanged OR stMetsStatus.stPCMStatus.bOpModeChanged, INT_TO_STRING(stMachineConfig.nMaximumOACFiles), '0'), strString6 := ' ', strString7 := 'FALSE FALSE'),
    START := fbMaintainDeleteTime.bOutput AND nActivateBitWord.6 OR NOT (stMachineConfig.stProductionLine.sPCM = '') AND (stMetsStatus.stPCMStatus.bRSKUChanged OR stMetsStatus.stPCMStatus.bOpModeChanged) OR aManualMaintain[6],
    TMOUT := cONE_SECOND); // NT_StartProcess

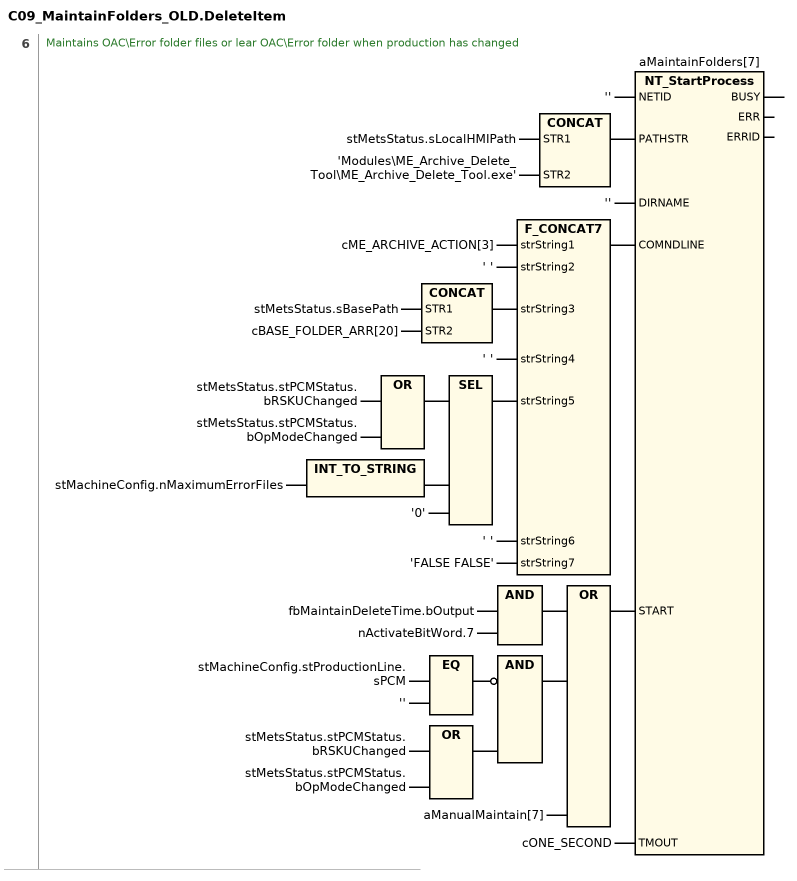
// NETWORK 6
// Maintains OAC\Error folder files or lear OAC\Error folder when production has changed
aMaintainFolders[7](
    NETID := '',
    PATHSTR := CONCAT(STR1 := stMetsStatus.sLocalHMIPath, STR2 := 'Modules\ME_Archive_Delete_Tool\ME_Archive_Delete_Tool.exe'),
    DIRNAME := '',
    COMNDLINE := F_CONCAT7(strString1 := cME_ARCHIVE_ACTION[3], strString2 := ' ', strString3 := CONCAT(STR1 := stMetsStatus.sBasePath, STR2 := cBASE_FOLDER_ARR[20]), strString4 := ' ', strString5 := SEL(stMetsStatus.stPCMStatus.bRSKUChanged OR stMetsStatus.stPCMStatus.bOpModeChanged, INT_TO_STRING(stMachineConfig.nMaximumErrorFiles), '0'), strString6 := ' ', strString7 := 'FALSE FALSE'),
    START := fbMaintainDeleteTime.bOutput AND nActivateBitWord.7 OR NOT (stMachineConfig.stProductionLine.sPCM = '') AND (stMetsStatus.stPCMStatus.bRSKUChanged OR stMetsStatus.stPCMStatus.bOpModeChanged) OR aManualMaintain[7],
    TMOUT := cONE_SECOND); // NT_StartProcess

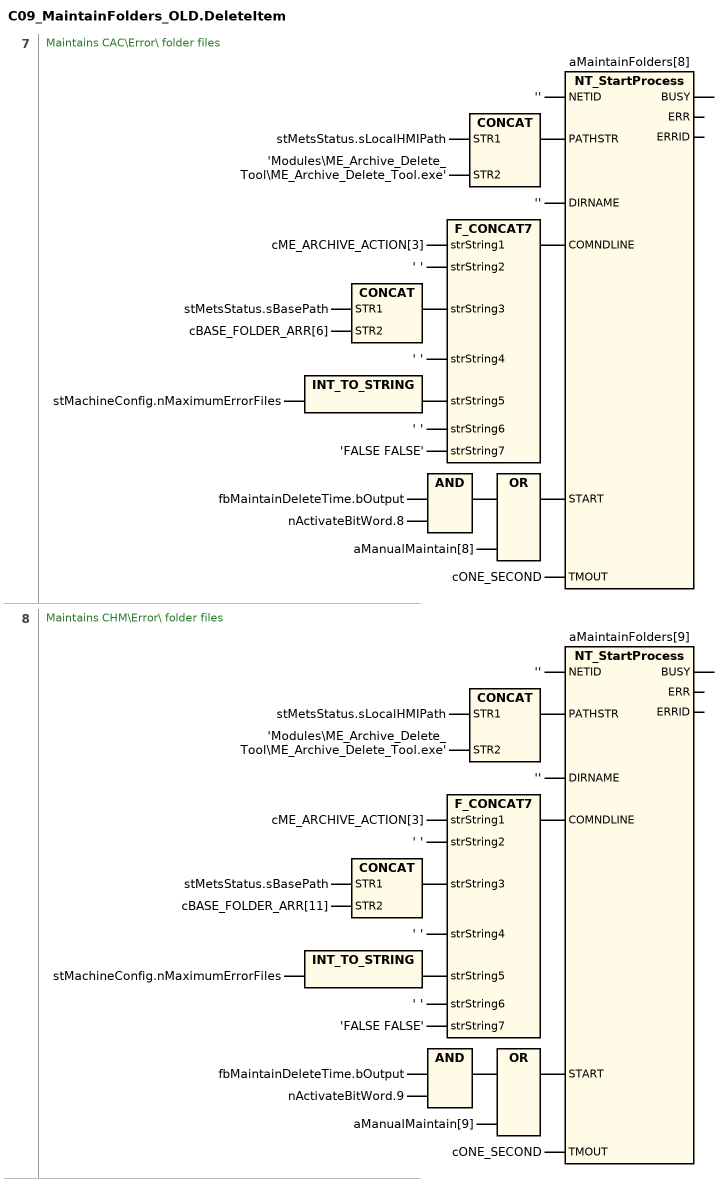
// NETWORK 7
// Maintains CAC\Error\ folder files
aMaintainFolders[8](
    NETID := '',
    PATHSTR := CONCAT(STR1 := stMetsStatus.sLocalHMIPath, STR2 := 'Modules\ME_Archive_Delete_Tool\ME_Archive_Delete_Tool.exe'),
    DIRNAME := '',
    COMNDLINE := F_CONCAT7(strString1 := cME_ARCHIVE_ACTION[3], strString2 := ' ', strString3 := CONCAT(STR1 := stMetsStatus.sBasePath, STR2 := cBASE_FOLDER_ARR[6]), strString4 := ' ', strString5 := INT_TO_STRING(stMachineConfig.nMaximumErrorFiles), strString6 := ' ', strString7 := 'FALSE FALSE'),
    START := fbMaintainDeleteTime.bOutput AND nActivateBitWord.8 OR aManualMaintain[8],
    TMOUT := cONE_SECOND); // NT_StartProcess

// NETWORK 8
// Maintains CHM\Error\ folder files
aMaintainFolders[9](
    NETID := '',
    PATHSTR := CONCAT(STR1 := stMetsStatus.sLocalHMIPath, STR2 := 'Modules\ME_Archive_Delete_Tool\ME_Archive_Delete_Tool.exe'),
    DIRNAME := '',
    COMNDLINE := F_CONCAT7(strString1 := cME_ARCHIVE_ACTION[3], strString2 := ' ', strString3 := CONCAT(STR1 := stMetsStatus.sBasePath, STR2 := cBASE_FOLDER_ARR[11]), strString4 := ' ', strString5 := INT_TO_STRING(stMachineConfig.nMaximumErrorFiles), strString6 := ' ', strString7 := 'FALSE FALSE'),
    START := fbMaintainDeleteTime.bOutput AND nActivateBitWord.9 OR aManualMaintain[9],
    TMOUT := cONE_SECOND); // NT_StartProcess

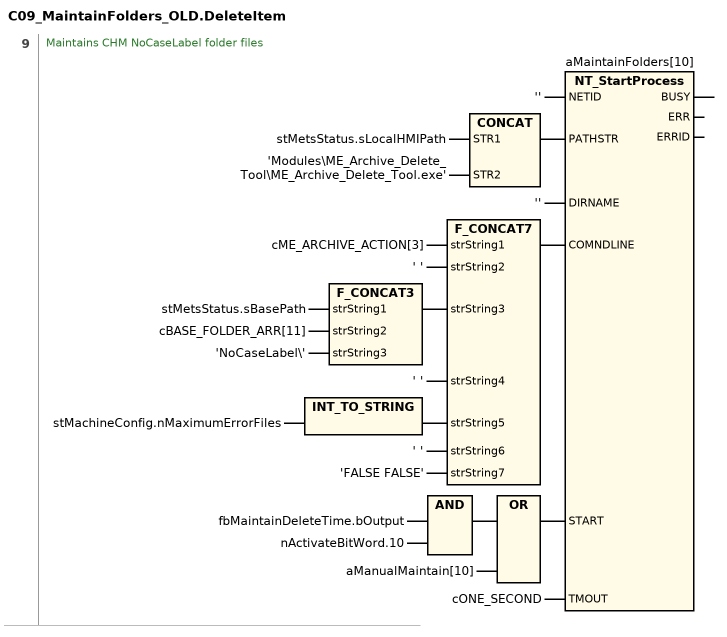
// NETWORK 9
// Maintains CHM NoCaseLabel folder files
aMaintainFolders[10](
    NETID := '',
    PATHSTR := CONCAT(STR1 := stMetsStatus.sLocalHMIPath, STR2 := 'Modules\ME_Archive_Delete_Tool\ME_Archive_Delete_Tool.exe'),
    DIRNAME := '',
    COMNDLINE := F_CONCAT7(strString1 := cME_ARCHIVE_ACTION[3], strString2 := ' ', strString3 := F_CONCAT3(strString1 := stMetsStatus.sBasePath, strString2 := cBASE_FOLDER_ARR[11], strString3 := 'NoCaseLabel\'), strString4 := ' ', strString5 := INT_TO_STRING(stMachineConfig.nMaximumErrorFiles), strString6 := ' ', strString7 := 'FALSE FALSE'),
    START := fbMaintainDeleteTime.bOutput AND nActivateBitWord.10 OR aManualMaintain[10],
    TMOUT := cONE_SECOND); // NT_StartProcess
END_ACTION

ACTION DeleteTime:
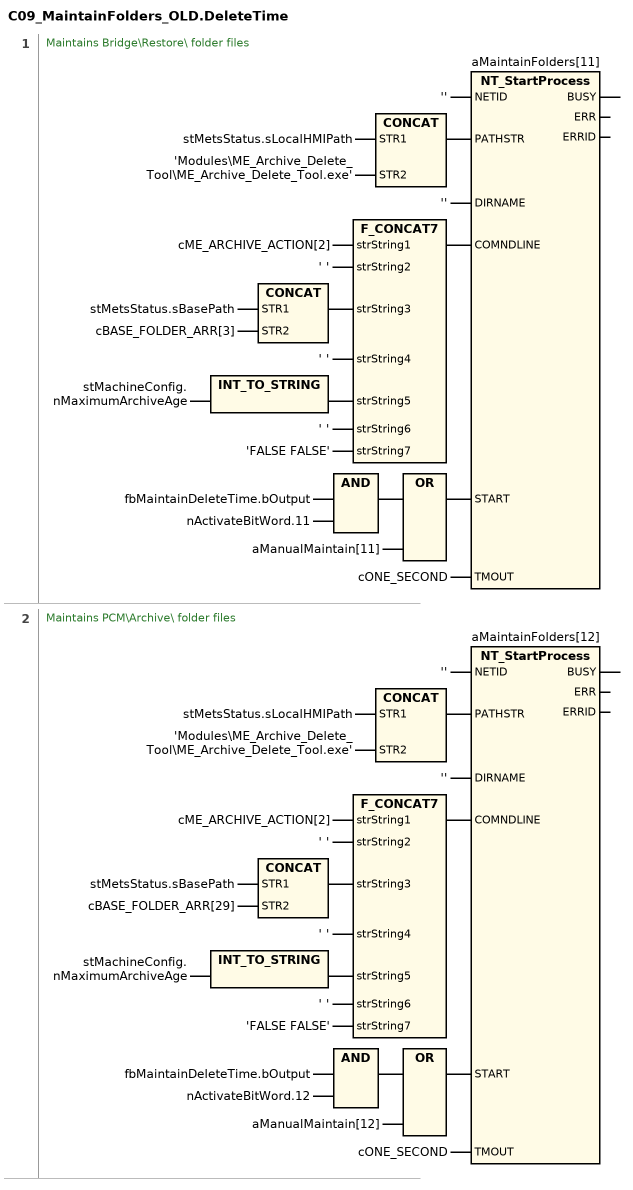
// NETWORK 1
// Maintains Bridge\Restore\ folder files
aMaintainFolders[11](
    NETID := '',
    PATHSTR := CONCAT(STR1 := stMetsStatus.sLocalHMIPath, STR2 := 'Modules\ME_Archive_Delete_Tool\ME_Archive_Delete_Tool.exe'),
    DIRNAME := '',
    COMNDLINE := F_CONCAT7(strString1 := cME_ARCHIVE_ACTION[2], strString2 := ' ', strString3 := CONCAT(STR1 := stMetsStatus.sBasePath, STR2 := cBASE_FOLDER_ARR[3]), strString4 := ' ', strString5 := INT_TO_STRING(stMachineConfig.nMaximumArchiveAge), strString6 := ' ', strString7 := 'FALSE FALSE'),
    START := fbMaintainDeleteTime.bOutput AND nActivateBitWord.11 OR aManualMaintain[11],
    TMOUT := cONE_SECOND); // NT_StartProcess

// NETWORK 2
// Maintains PCM\Archive\ folder files
aMaintainFolders[12](
    NETID := '',
    PATHSTR := CONCAT(STR1 := stMetsStatus.sLocalHMIPath, STR2 := 'Modules\ME_Archive_Delete_Tool\ME_Archive_Delete_Tool.exe'),
    DIRNAME := '',
    COMNDLINE := F_CONCAT7(strString1 := cME_ARCHIVE_ACTION[2], strString2 := ' ', strString3 := CONCAT(STR1 := stMetsStatus.sBasePath, STR2 := cBASE_FOLDER_ARR[29]), strString4 := ' ', strString5 := INT_TO_STRING(stMachineConfig.nMaximumArchiveAge), strString6 := ' ', strString7 := 'FALSE FALSE'),
    START := fbMaintainDeleteTime.bOutput AND nActivateBitWord.12 OR aManualMaintain[12],
    TMOUT := cONE_SECOND); // NT_StartProcess

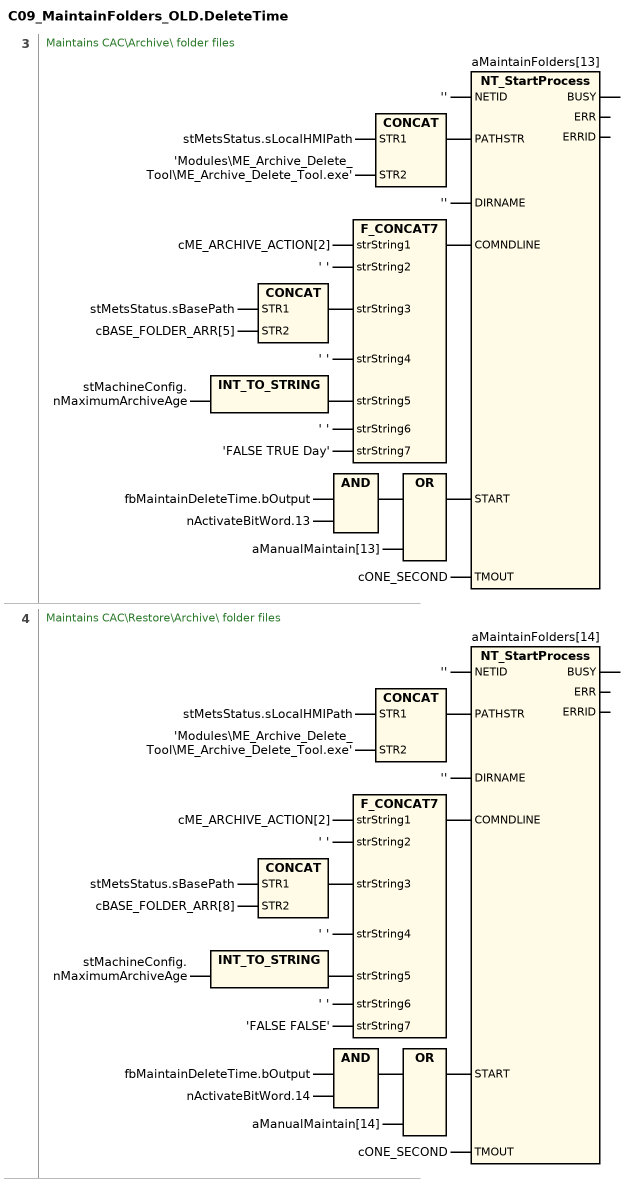
// NETWORK 3
// Maintains CAC\Archive\ folder files
aMaintainFolders[13](
    NETID := '',
    PATHSTR := CONCAT(STR1 := stMetsStatus.sLocalHMIPath, STR2 := 'Modules\ME_Archive_Delete_Tool\ME_Archive_Delete_Tool.exe'),
    DIRNAME := '',
    COMNDLINE := F_CONCAT7(strString1 := cME_ARCHIVE_ACTION[2], strString2 := ' ', strString3 := CONCAT(STR1 := stMetsStatus.sBasePath, STR2 := cBASE_FOLDER_ARR[5]), strString4 := ' ', strString5 := INT_TO_STRING(stMachineConfig.nMaximumArchiveAge), strString6 := ' ', strString7 := 'FALSE TRUE Day'),
    START := fbMaintainDeleteTime.bOutput AND nActivateBitWord.13 OR aManualMaintain[13],
    TMOUT := cONE_SECOND); // NT_StartProcess

// NETWORK 4
// Maintains CAC\Restore\Archive\ folder files
aMaintainFolders[14](
    NETID := '',
    PATHSTR := CONCAT(STR1 := stMetsStatus.sLocalHMIPath, STR2 := 'Modules\ME_Archive_Delete_Tool\ME_Archive_Delete_Tool.exe'),
    DIRNAME := '',
    COMNDLINE := F_CONCAT7(strString1 := cME_ARCHIVE_ACTION[2], strString2 := ' ', strString3 := CONCAT(STR1 := stMetsStatus.sBasePath, STR2 := cBASE_FOLDER_ARR[8]), strString4 := ' ', strString5 := INT_TO_STRING(stMachineConfig.nMaximumArchiveAge), strString6 := ' ', strString7 := 'FALSE FALSE'),
    START := fbMaintainDeleteTime.bOutput AND nActivateBitWord.14 OR aManualMaintain[14],
    TMOUT := cONE_SECOND); // NT_StartProcess

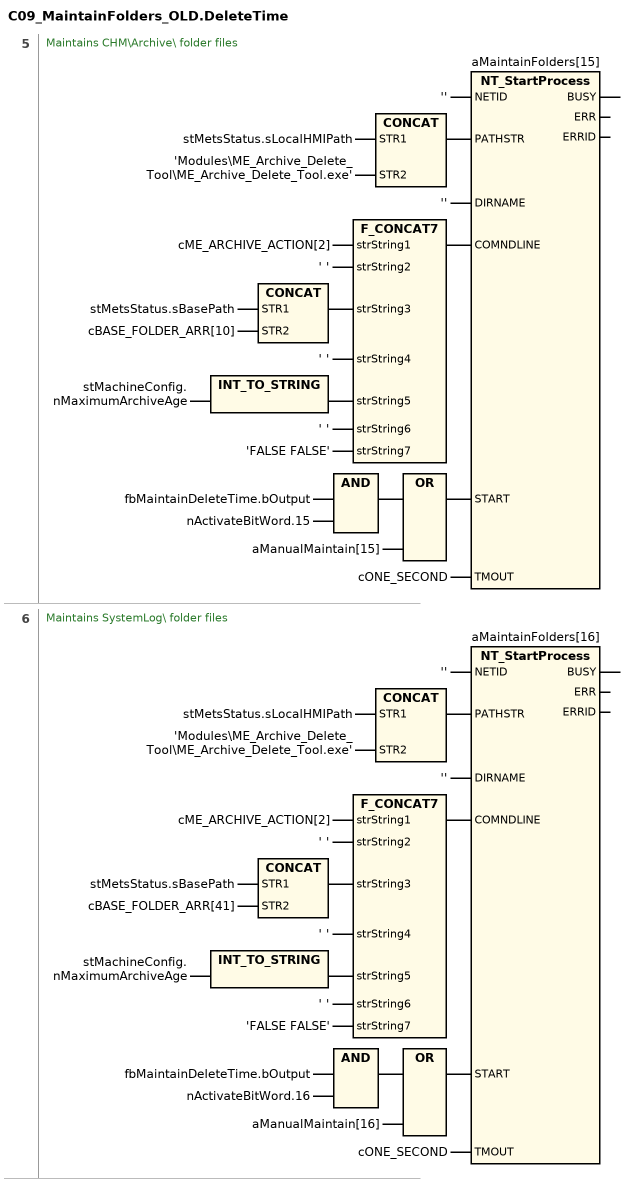
// NETWORK 5
// Maintains CHM\Archive\ folder files
aMaintainFolders[15](
    NETID := '',
    PATHSTR := CONCAT(STR1 := stMetsStatus.sLocalHMIPath, STR2 := 'Modules\ME_Archive_Delete_Tool\ME_Archive_Delete_Tool.exe'),
    DIRNAME := '',
    COMNDLINE := F_CONCAT7(strString1 := cME_ARCHIVE_ACTION[2], strString2 := ' ', strString3 := CONCAT(STR1 := stMetsStatus.sBasePath, STR2 := cBASE_FOLDER_ARR[10]), strString4 := ' ', strString5 := INT_TO_STRING(stMachineConfig.nMaximumArchiveAge), strString6 := ' ', strString7 := 'FALSE FALSE'),
    START := fbMaintainDeleteTime.bOutput AND nActivateBitWord.15 OR aManualMaintain[15],
    TMOUT := cONE_SECOND); // NT_StartProcess

// NETWORK 6
// Maintains SystemLog\ folder files
aMaintainFolders[16](
    NETID := '',
    PATHSTR := CONCAT(STR1 := stMetsStatus.sLocalHMIPath, STR2 := 'Modules\ME_Archive_Delete_Tool\ME_Archive_Delete_Tool.exe'),
    DIRNAME := '',
    COMNDLINE := F_CONCAT7(strString1 := cME_ARCHIVE_ACTION[2], strString2 := ' ', strString3 := CONCAT(STR1 := stMetsStatus.sBasePath, STR2 := cBASE_FOLDER_ARR[41]), strString4 := ' ', strString5 := INT_TO_STRING(stMachineConfig.nMaximumArchiveAge), strString6 := ' ', strString7 := 'FALSE FALSE'),
    START := fbMaintainDeleteTime.bOutput AND nActivateBitWord.16 OR aManualMaintain[16],
    TMOUT := cONE_SECOND); // NT_StartProcess

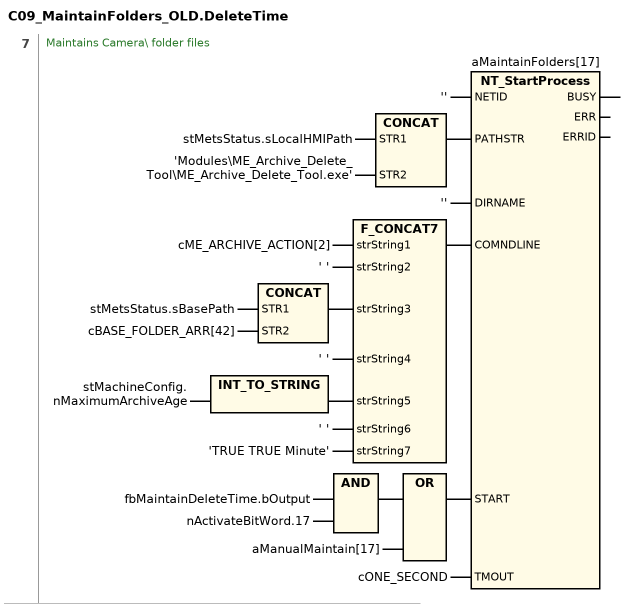
// NETWORK 7
// Maintains Camera\ folder files
aMaintainFolders[17](
    NETID := '',
    PATHSTR := CONCAT(STR1 := stMetsStatus.sLocalHMIPath, STR2 := 'Modules\ME_Archive_Delete_Tool\ME_Archive_Delete_Tool.exe'),
    DIRNAME := '',
    COMNDLINE := F_CONCAT7(strString1 := cME_ARCHIVE_ACTION[2], strString2 := ' ', strString3 := CONCAT(STR1 := stMetsStatus.sBasePath, STR2 := cBASE_FOLDER_ARR[42]), strString4 := ' ', strString5 := INT_TO_STRING(stMachineConfig.nMaximumArchiveAge), strString6 := ' ', strString7 := 'TRUE TRUE Minute'),
    START := fbMaintainDeleteTime.bOutput AND nActivateBitWord.17 OR aManualMaintain[17],
    TMOUT := cONE_SECOND); // NT_StartProcess
END_ACTION

ACTION ShiftActivationBit:
IF fbMaintainDeleteTime.bOutput	THEN
	IF nActivateBitWord = 0 THEN
		nActivateBitWord := 1;
	ELSE
		nActivateBitWord :=SHL(nActivateBitWord,1);
	END_IF
END_IF
END_ACTION

END_PROGRAM

// ---- POUs/_Exclude/v2/FB_CAC_RestoreOAC.TcPOU
(* reads CAC files from CAC folder and archives OAC file *)
FUNCTION_BLOCK FB_CAC_RestoreOAC
VAR_INPUT
	bExecute					: BOOL;		(* set TRUE to check for CAC files to be restored *)
	ePackAggregationMode	: E_SYSTEM_PackAggregationMode ;
	sLocalOCVPath				: STRING(255);	(* TEMP folder path *)
	sLocalOACPath				: STRING(255);	(* path to OAC folder *)
	sLocalCACPath				: STRING(255);	(* path to CAC Watch folder *)
	nPacksPerOuter			: INT;
	nPackPos1					: INT 	:=1;
	nPackPos2					: INT	:=2;
	bUseInterimCodeForValidation	 : BOOL;
END_VAR
VAR_IN_OUT
	stCodeInfo_Pack			: ST_CodeInfo;
	stCodeInfo_Intermediate		: ST_CodeInfo;
	stCodeInfo_Case			: ST_CodeInfo;
END_VAR
VAR_OUTPUT
	bDone 					: BOOL;		(* TRUE = OAC restore complete *)
	bBusy 					: BOOL;		(* TRUE = OAC restore active *)
	bError 					: BOOL;		(* TRUE = OAC restore error *)
	nErrorID					: UDINT;	(* error code *)
	sCACRestored				: STRING;
	nOCVFilesRestored			: UDINT;
	nOACFilesRestored			: UDINT;
	nCACFilesRestored			: UDINT;
END_VAR
VAR
	fbExecute					: R_TRIG;
	eState					: E_CAC_State;
	eErrorState				: E_CAC_State;
	stOCVPackStatus			: ST_OUTER_Status;
	stCACData					: ST_CAC_Data;
	fbFindCACFile				: FB_EnumFindFileEntry;
	eCmdType				: E_EnumCmdType;
	strOACFile				: T_OAC_Filename;
	strCACFile				: T_CAC_Filename;
	fbReadCACData			: FB_XmlSrvRead;
	nOuterIndex				: INT;
	fbWriteOACFile			: FB_OAC_WriteFile;
	nOCVindex				: INT;
	fbWriteOCVFile			: FB_OCV_WriteFile;
	fbCopyFile				: FB_FILE_CopyByByte;
	fbDeleteFile				: FB_FileDelete;

	aOCVFileCodeName			: ARRAY[1..2] OF T_MaxString;

	bAggregationCodes1Valid			: BOOL;
	bAggregationCodes2Valid			: BOOL;
END_VAR

(* monitor bExecute for rising edge *)
fbExecute(CLK := bExecute);

CASE eState OF

	(* idle *)
	E_CAC_IDLE:

		(* rising edge of bExecute *)
		IF fbExecute.Q = TRUE THEN

			(* update outputs *)
			bDone := FALSE;
			bBusy := TRUE;
			bError := FALSE;
			nErrorID := 0;

			nOuterIndex	:=0;
			nOCVindex	:=0;

			(* clear outputs *)
			nOCVFilesRestored :=0;
			nOACFilesRestored := 0;
			nCACFilesRestored := 0;

			(* initiliase vars *)
			eCmdType := eEnumCmd_First;
			eErrorState := eState;
			sCACRestored	:= '';
			MEMSET(ADR(strCACFile), 16#00, SIZEOF(strCACFile));
			MEMSET(ADR(aOCVFileCodeName), 16#00, SIZEOF(aOCVFileCodeName));

			eState := E_CAC_FINDFILE;

		(* bExecute has been reset *)
		ELSIF bExecute = FALSE THEN

			(* clear outputs *)
			bDone := FALSE;
			bBusy := FALSE;
			bError := FALSE;
			nErrorID := 0;
		END_IF


	(* build list of CAC files to be restored *)
	E_CAC_FINDFILE:

		(* build list *)
		fbFindCACFile(
			sNetId		:= '',
			sPathName	:= F_CONCAT3(sLocalCACPath, 'Restore\', 'CAC_*.xml'),
			eCmd		:= eCmdType,
			bExecute	:= TRUE,
			tTimeout	:= T#5s
		);

		(* find CAC file complete *)
		IF fbFindCACFile.bBusy = FALSE THEN

			(* find CAC file completed OK *)
			IF fbFindCACFile.bError = FALSE THEN

				(* end of CAC file list *)
				IF fbFindCACFile.bEOE = TRUE OR eCmdType = eEnumCmd_Abort THEN

					eState := E_CAC_DONE;

				(* next CAC file *)
				ELSE

					(* next CAC file *)
					strCACFile := fbFindCACFile.stFindFile.sFileName;
					sCACRestored := MID(strCACFile,  stCodeInfo_Case.stSerialCode.nCodeLength,stCodeInfo_Case.stSerialCode.nCodeStartPos + LEN('CAC_'));
					eCmdType := eEnumCmd_Next;
					MEMSET(ADR(stCACData), 16#00, SIZEOF(stCACData));

					eState := E_CAC_READDATA;
				END_IF

			(* find CAC file error *)
			ELSE

				bError := TRUE;
				nErrorID := fbFindCACFile.nErrID;
				eErrorState := eState;

				eState := E_CAC_DONE;
			END_IF

			(* close off fbFindCACFile *)
			fbFindCACFile(bExecute := FALSE);
		END_IF


	(* load CAC file *)
	E_CAC_READDATA:

		(* load CAC data *)
		fbReadCACData(
			sNetId		:= '',
			ePath		:= PATH_GENERIC,
			nMode		:= XMLSRV_SKIPMISSING,
			pSymAddr	:= ADR(stCACData),
			cbSymSize	:= SIZEOF(stCACData),
			sFilePath	:= F_CONCAT3(sLocalCACPath, 'Restore\', strCACFile),
			sXPath		:= '/Case',
			bExecute	:= TRUE,
			tTimeout	:= T#1s
		);

		(* load CAC data complete *)
		IF fbReadCACData.bBusy = FALSE THEN

			(* load CAC data completed OK *)
			IF fbReadCACData.bError = FALSE THEN

				(* first Outer *)
				nOuterIndex := 1;

				eState := E_CAC_WRITEDATA;

			(* load CAC data error *)
			ELSE

				bError := TRUE;
				nErrorID := fbReadCACData.nErrId;
				eErrorState := eState;

				eState := E_CAC_FINDFILE;
			END_IF

			(* close off fbReadCACData *)
			fbReadCACData(bExecute := FALSE);
		END_IF


	(* create OAC files *)
	E_CAC_WRITEDATA:

		FOR nOCVindex :=1 TO stCACData.Outer[nOuterIndex].NumberOfPacks DO
			stCACData.Outer[nOuterIndex].PackCodeStatus[nOCVindex].8 := TRUE;
		END_FOR

		fbWriteOACFile(
			bExecute			:= TRUE,
			sLocalOACPath	:= sLocalOACPath,
			stOACData			:= stCACData.Outer[nOuterIndex],
			sOACFile		=> strOACFile
		);

		(* create folder complete *)
		IF fbWriteOACFile.bDone = TRUE THEN

			(* write OAC file completed OK *)
			IF fbWriteOACFile.bError = FALSE THEN

				(* total OAC files restored *)
				nOACFilesRestored := nOACFilesRestored + 1;
			END_IF

			eState := E_CAC_CREATEOCVDATA;

			(* close off fbWriteOACFile *)
			fbWriteOACFile(bExecute := FALSE);
		END_IF
(* write OCVC file *)
	E_CAC_CREATEOCVDATA:

			bAggregationCodes1Valid := FALSE;
			bAggregationCodes2Valid := FALSE;

			stOCVPackStatus.stOACData := stCACData.Outer[nOuterIndex];
			stOCVPackStatus.nTriggerID :=9999;

			FOR nOCVindex :=1 TO stOCVPackStatus.stOACData.NumberOfPacks DO

				IF	stOCVPackStatus.stOACData.PackCode[nOCVindex] <> '' THEN
					(*stOCVPackStatus.stOACData.PackRejectCode[nOCVindex] := 'OK';
					stOCVPackStatus.stOACData.PackRejectID[nOCVindex] := 0;
					stOCVPackStatus.aPackSUPIResult[nOCVindex]:= nSUPIIdentyfication;*)
					stOCVPackStatus.aOACPackStatus[nOCVindex] :=5;
				ELSE
					(*stOCVPackStatus.stOACData.PackRejectCode[nOCVindex] := 'Pack code(s)  no read';
					stOCVPackStatus.stOACData.PackRejectID[nOCVindex] := 101;*)
					stOCVPackStatus.aOACPackStatus[nOCVindex] :=0;
					(*stOCVPackStatus.aPackSUPIResult[nOCVindex]:= -2;*)
				END_IF

				stOCVPackStatus.aPackCodeFilledIn[nOCVindex] := E_PACK_CODERESTOREDCAC;
				stOCVPackStatus.aPackCodes[nOCVindex].sBuffer[1].strCode := stOCVPackStatus.stOACData.PackCode[nOCVindex];
				stOCVPackStatus.aPackCodes[nOCVindex].sBuffer[1].nStatus := stOCVPackStatus.aOACPackStatus[nOCVindex];
				stOCVPackStatus.aPackCodes[nOCVindex].sBuffer[1].nStringSize := LEN(stOCVPackStatus.stOACData.PackCode[nOCVindex]);
				stOCVPackStatus.aPackCodes[nOCVindex].sBuffer[2].strCode := stOCVPackStatus.stOACData.PackCode[nOCVindex];
				stOCVPackStatus.aPackCodes[nOCVindex].sBuffer[2].nStatus := stOCVPackStatus.aOACPackStatus[nOCVindex];
				stOCVPackStatus.aPackCodes[nOCVindex].sBuffer[2].nStringSize := LEN(stOCVPackStatus.stOACData.PackCode[nOCVindex]);
			END_FOR

		eState := E_CAC_WRITEOCVDATA;

	E_CAC_WRITEOCVDATA:

		aOCVFileCodeName[1]	:=	F_CodeToHex(F_CODE_GetItem(stOCVPackStatus.stOACData.AggregationCodes[1] , eCodeAIType.SerialCode,
																				SEL(bUseInterimCodeForValidation, stCodeInfo_Pack, stCodeInfo_Intermediate)));
		aOCVFileCodeName[2]	:=	F_CodeToHex(F_CODE_GetItem(stOCVPackStatus.stOACData.AggregationCodes[2] , eCodeAIType.SerialCode,   stCodeInfo_Pack)); (*no reason to have 2 diffrent intermediate codes*)

		IF F_InvalidateASCIIChar(aOCVFileCodeName[1]) =	0 	THEN bAggregationCodes1Valid := nPackPos1 <> 0 OR  bUseInterimCodeForValidation;  	END_IF
		IF F_InvalidateASCIIChar(aOCVFileCodeName[2]) =	0 	THEN bAggregationCodes2Valid := nPackPos2 <> 0; 		END_IF

		(* write OCV file *)
		fbWriteOCVFile(
			bExecute					:= TRUE,
			sTargetPath				:= sLocalOCVPath,
			ePackAggregationMode	:= ePackAggregationMode,
			nPacksPerOuter			:= nPacksPerOuter,
			aOCVFileCodeName		:= aOCVFileCodeName,  (*strAggregationCodes is a table*)
			bSkipWriteFile1			:= NOT bAggregationCodes1Valid,
			bSkipWriteFile2			:= NOT bAggregationCodes2Valid,
			stOCVPackStatus			:= stOCVPackStatus
			);


		(*IF F_PACK_ValidateCodeASCII(F_CODE_GetItem(stOCVPackStatus.stOACData.PackCode[nPackPos1], eCodeAIType.SerialCode, stMachineConfig.stCodeInfo_Pack)) =
						stMachineConfig.stCodeInfo_Pack.stSerialCode.nCodeLength 	 THEN bPackCode1Valid := TRUE;  	END_IF

		IF	F_PACK_ValidateCodeASCII(F_CODE_GetItem(stOCVPackStatus.stOACData.PackCode[nPackPos2], eCodeAIType.SerialCode, stMachineConfig.stCodeInfo_Pack)) =
						stMachineConfig.stCodeInfo_Pack.stSerialCode.nCodeLength 	THEN bPackCode2Valid := TRUE; 	END_IF

		(* write OCV file *)
		fbWriteOCVFile(
			bExecute				:= TRUE,
			strTargetPath			:= sLocalOCVPath,
			nPacksPerOuter		:= nPacksPerOuter,
			nPackPos1			:= nPackPos1,
			bSkipWriteFile1		:= NOT bPackCode1Valid,
			nPackPos2			:= nPackPos2,
			bSkipWriteFile2		:= NOT bPackCode2Valid,
			stOCVPackStatus		:= stOCVPackStatus
			);*)

		(* write OCV file complete *)
		IF fbWriteOCVFile.bDone = TRUE THEN

			(* write OCV file completed OK *)
			IF fbWriteOCVFile.bError = FALSE THEN

				nOCVFilesRestored	:= nOCVFilesRestored +2;

			END_IF

			nOuterIndex := nOuterIndex + 1;
			(* last Outer *)
			IF nOuterIndex > stCACData.NumberOfOuters THEN

				(* total CAC files restored *)
				nCACFilesRestored := nCACFilesRestored + 1;

				eState := E_CAC_COPYFILE;
			(* not last Outer *)
			ELSE

			eState := E_CAC_WRITEDATA;
			END_IF

			(* close off fbWriteOCVFile*)
			fbWriteOCVFile(bExecute := FALSE);
		END_IF
	(* copy CAC file to archive folder *)
	E_CAC_COPYFILE:

		(* copy CAC file *)
		fbCopyFile(
			bExecute		:= TRUE,
			strPathSource	:= F_CONCAT3(sLocalCACPath, 'Restore\', strCACFile),
			strPathTarget	:= F_CONCAT3(sLocalCACPath, 'Restore\Archive\', strCACFile),
			strFileName		:= '',
			tTimeout		:= T#1s
		);

		(* copy file complete *)
		IF fbCopyFile.bBusy = FALSE THEN

			(* copy file completed OK or CAC file not found *)
			IF fbCopyFile.bError = FALSE THEN

				eState := E_CAC_DELETEFILE;

			(* copy command error *)
			ELSE

				bError := TRUE;
				nErrorID := fbCopyFile.nErrorId;
				eErrorState := eState;

				eState := E_CAC_DELETEFILE;
			END_IF

			(* close off fbCopyFile *)
			fbCopyFile(bExecute := FALSE);
		END_IF

	(* delete CAC file *)
	E_CAC_DELETEFILE:

		(* delete file *)
		fbDeleteFile(
			sNetId		:= '',
			sPathName	:= F_CONCAT3(sLocalCACPath, 'Restore\', strCACFile),
			ePath		:= PATH_GENERIC,
			bExecute	:= TRUE,
			tTimeout	:= T#1s
		);

		(* delete file complete *)
		IF fbDeleteFile.bBusy = FALSE THEN

			eState := E_CAC_FINDFILE;

			(* close off fbDeleteFile *)
			fbDeleteFile(bExecute  := FALSE);
		END_IF


	(* complete *)
	E_CAC_DONE:

		(* update outputs *)
		bBusy := FALSE;
		bDone := TRUE;

		eState := E_CAC_IDLE;


(* unknown state *)
ELSE

	eState := E_CAC_IDLE;
END_CASE

END_FUNCTION_BLOCK

// ---- POUs/_Exclude/OAC FBs/FB_OAC_WriteFile.TcPOU
FUNCTION_BLOCK FB_OAC_WriteFile
VAR_INPUT
	bExecute					: BOOL;			(* scan for valid Outer in arrOuterStatus *)
	sLocalOACPath				: STRING(50);	(* target folder for OAC file *)
	bInvalidOAC				: BOOL;
	bOACDupBacroceFound	: BOOL;
	bOACDupPacksFound		: BOOL;
	stCTDateTime				: ST_SYSTEM_DateTime;
	stOACData					: ST_OAC_Data;
	tTimeout					: TIME := cHALF_SECOND;
END_VAR
VAR_OUTPUT
	bDone				: BOOL;			(* TRUE = write OAC file complete *)
	bBusy				: BOOL;			(* TRUE = write OAC file in progress *)
	bError				: BOOL;			(* TRUE = write OAC file error *)
	nErrorID			: UDINT;		(* error ID *)
	sOACFile			: T_OAC_Filename;	(* OAC file name *)
	sLastCretedFile		: T_MaxString;
END_VAR
VAR
	fbExecute			: R_TRIG;
	eState				: E_OUTER_State;
	eErrorState			: E_OUTER_State;
	fbBuildOACData		: FB_OAC_BuildXMLData;
	fbCreateFolder		: FB_CreateDir;
	fbWriteFile			: FB_FILE_WriteByByte;
	sTargetPath			: STRING(50);
	aDebugOACFile			: ARRAY[1..10] OF  T_OAC_Filename;	(* OAC file name *)
	nCounter :UDINT;
END_VAR

(* monitor bExecute for rising edge *)
fbExecute(CLK := bExecute);

CASE eState OF

	(* idle *)
	E_OUTER_IDLE:

		(* rising edge on bExecute *)
		IF fbExecute.Q = TRUE THEN

			(* update outputs *)
			bDone := FALSE;
			bBusy := TRUE;
			bError := FALSE;
			nErrorID := 0;

			sLastCretedFile := '';

		(*	bInvalidOAC	:= TRUE; - mod done for test only*)

			(* generate OAC file name and clear data for last OAC file *)

			IF bInvalidOAC THEN
				sTargetPath :=CONCAT(sLocalOACPath,'Error\' );

				IF bOACDupPacksFound THEN
					 sOACFile := F_CONCAT5('DUP_PK_OAC_', F_OUTER_BarcodeToHex(stOACData.Barcode),'_' ,  F_SYSTEM_SystemTimeToCHM_Header(stCTDateTime.sSystemTime),'.xml');
				ELSIF bOACDupBacroceFound THEN
					sOACFile := F_CONCAT5('DUP_BC_OAC_', F_OUTER_BarcodeToHex(stOACData.Barcode),'_' ,  F_SYSTEM_SystemTimeToCHM_Header(stCTDateTime.sSystemTime),'.xml');
				ELSE
					sOACFile := F_CONCAT5('ERR_OAC_', F_OUTER_BarcodeToHex(stOACData.Barcode),'_' ,  F_SYSTEM_SystemTimeToCHM_Header(stCTDateTime.sSystemTime),'.xml');
				END_IF
			ELSE
				sTargetPath := sLocalOACPath;
				sOACFile := F_CONCAT3('OAC_', F_OUTER_BarcodeToHex(stOACData.Barcode), '.xml');
			END_IF

			(*strOACFile := F_CONCAT3('OAC_', F_SCANNER_RemoveAIBrackets(stOACData.Barcode), '.xml');*)

			nCounter := nCounter +1;
			MEMMOVE(ADR(aDebugOACFile[2]), ADR(aDebugOACFile[1]), SIZEOF(aDebugOACFile)-SIZEOF(aDebugOACFile[1]));
			aDebugOACFile[1] := F_CONCAT3(sOACFile,'_', UDINT_TO_STRING(nCounter));

			eState := E_OUTER_BUILDXMLIMAGE;

		(* disabled *)
		ELSIF bExecute = FALSE THEN

			(* update outputs *)
			bDone := FALSE;
			bBusy := FALSE;
			(*bError := FALSE;
			nErrorID := 0;*)
		END_IF


	(* build OAC image in XML format *)
	E_OUTER_BUILDXMLIMAGE:

		(* build OAC data *)
		fbBuildOACData(
			bExecute		:= TRUE,
			bAddXMLHeader	:= TRUE,
			nTabIndent		:= 0,
			nOuterIndex		:= 0,
			stOACData		:= stOACData
		);

		(* build OAC data complete *)
		IF fbBuildOACData.bDone = TRUE THEN

			eState := E_OUTER_CREATEERRORFOLDER;

			(* close off fbBuildOACData *)
			fbBuildOACData(bExecute := FALSE);
		END_IF

(***************************************************************************)

	(* create folders *)
	E_OUTER_CREATEERRORFOLDER:

		(* create date archive folder *)
		fbCreateFolder(
			sNetId		:= '',
			sPathName	:= sTargetPath,
			ePath		:= PATH_GENERIC,
			bExecute	:= TRUE,
			tTimeout	:= T#1s
		);

		(* create folder complete *)
		IF fbCreateFolder.bBusy = FALSE THEN

			(* create folder completed OK or folder already exists *)
			IF fbCreateFolder.bError = FALSE OR (fbCreateFolder.bError = TRUE AND fbCreateFolder.nErrId = 16#70C) THEN

				eState := E_OUTER_WRITEXMLIMAGE;
			(* create folder error *)
			ELSE

				(* update outputs *)
				bError := TRUE;
				nErrorID := fbCreateFolder.nErrId;
				eErrorState := eState;

				eState := E_OUTER_DONE;
			END_IF

			(* close off fbCreateFolder *)
			fbCreateFolder(bExecute := FALSE);
		END_IF

(***************************************************************************)
	(* write OAC image *)
	E_OUTER_WRITEXMLIMAGE:

		(* write XML template to file *)
		fbWriteFile(
			bExecute	:= TRUE,
			pSourceAddr	:= ADR(fbBuildOACData.arrOACImage),
			nSourceSize	:= fbBuildOACData.nOACByte,
			strPathFile	:= CONCAT(sTargetPath, sOACFile),
			tTimeout	:= tTimeout
		);

		(* file write complete *)
		IF fbWriteFile.bDone = TRUE THEN

			(* file write completed OK *)
			IF fbWriteFile.bError = FALSE THEN

				sLastCretedFile := sOACFile;

			(* file write error *)
			ELSE

				bError := TRUE;
				nErrorID := fbWriteFile.nErrorID;
				eErrorState := eState;
			END_IF

			eState := E_OUTER_DONE;

			(* close of fbWriteFile *)
			fbWriteFile(bExecute := FALSE);
		END_IF


	(* OAC file complete *)
	E_OUTER_DONE:

		(* update outputs *)
		bDone := TRUE;
		bBusy := FALSE;

		eState := E_OUTER_IDLE;


(* unknown state *)
ELSE

	eState := E_OUTER_IDLE;
END_CASE

END_FUNCTION_BLOCK

// ---- POUs/_Exclude/OAC FBs/FB_OAC_BuildXMLData.TcPOU
FUNCTION_BLOCK FB_OAC_BuildXMLData
VAR_INPUT
	bExecute			: BOOL;
	bAddXMLHeader	: BOOL;
	nTabIndent		: BYTE;
	nOuterIndex		: INT;		(* Outer index when building for CAC file *)
	stOACData			: ST_OAC_Data;
END_VAR
VAR_OUTPUT
	bDone			: BOOL;
	nOACByte			: INT;		(* total bytes for OAC template *)
	arrOACImage		: ARRAY[0..20000] OF BYTE;
	bBufferOverflow	: BOOL;
END_VAR
VAR
	fbExecute			: R_TRIG;
	strPrefix			: T_MaxString; (*T_Char. strPrefix is assigned T_MaxString so T-Char will casue *)
	strString			: T_MaxString;
	nStringLen		: INT;
	nMaxOACImageSize	: UINT;
	nControlSize		: UINT;
	nMaxPackIndex	: INT;
	nPackIndex		: INT;
END_VAR

(* rising edge of bExecute *)
fbExecute(CLK := bExecute);


(* rising edge of bExecute *)
IF fbExecute.Q = TRUE THEN

	(* update outputs *)
	bDone := FALSE;
	bBufferOverflow	:=FALSE;

	(* clear output array and reset byte counter *)
	MEMSET(ADR(arrOACImage), 16#00, SIZEOF(arrOACImage));
	nOACByte := 0;
	nControlSize := 0;
	nMaxOACImageSize := SIZEOF(arrOACImage);

	(* XML header required *)
	IF bAddXMLHeader = TRUE THEN

		(* no prefix required, include XML header *)
		strString := cXML_HEADER;
		nStringLen := LEN(strString);
		MEMMOVE(ADR(arrOACImage[nOACByte]), ADR(strString), nStringLen);
		nOACByte := nOACByte + nStringLen;
		nControlSize := nOACByte;

		(* <Comment> tag *)
		strString := '<!--File OAC builder. Version 2.2.000 Relase 06.09.2022 PTR -->$R$N';
		AppendImageData();

	END_IF

	(* tab indent required *)
	IF nTabIndent > 0 THEN

		(* generate strPrefix with specified number of tabs *)
		strPrefix := F_StringAddPrefix('$T', nTabIndent, '$T');

	(* no tab index required *)
	ELSE

		(* clear strPrefix *)
		strPrefix := '';
	END_IF

	(* output is for CAC file *)
	IF nOuterIndex > 0 THEN

		(* <Outer index="xx"> tag *)
		strString := F_CONCAT4(strPrefix, '<Outer index="', INT_TO_STRING(nOuterIndex), '">$R$N');
		AppendImageData();

	(* output is for OAC file *)
	ELSE

		(* <Outer> tag *)
		strString := CONCAT(strPrefix, '<Outer>$R$N');
		AppendImageData();

	END_IF

	(* <Barcode> field *)
	strString := F_CONCAT4(strPrefix, '$T<Barcode><![CDATA[', stOACData.Barcode,']]></Barcode>$R$N');
	AppendImageData();

	(* <ProductionDate> field *)
	strString := F_CONCAT4(strPrefix, '$T<ProductionDate>', stOACData.ProductionDate, '</ProductionDate>$R$N');
	AppendImageData();

	(* <ProductionTime> field *)
	strString := F_CONCAT4(strPrefix, '$T<ProductionTime>', stOACData.ProductionTime, '</ProductionTime>$R$N');
	AppendImageData();

	(* <ProductionTimeOffset> field *)
	strString := F_CONCAT4(strPrefix, '$T<ProductionTimeOffset>', stOACData.ProductionTimeOffset, '</ProductionTimeOffset>$R$N');
	AppendImageData();

	(* <ProductionTimeStamp> field *)
	strString := F_CONCAT4(strPrefix, '$T<OuterTimeStamp>', stOACData.OuterTimeStamp, '</OuterTimeStamp>$R$N');
	AppendImageData();

	(* <ProductionTimeStamp> field *)
	strString := F_CONCAT4(strPrefix, '$T<PackTimeStamp>', stOACData.PackTimeStamp, '</PackTimeStamp>$R$N');
	AppendImageData();

	(* <RetailSKU> field *)
	strString := F_CONCAT4(strPrefix, '$T<RetailSKU>', stOACData.RetailSKU, '</RetailSKU>$R$N');
	AppendImageData();

	(* <OuterMachine> tag *)
	strString := CONCAT(strPrefix, '$T<OuterMachine>$R$N');
	AppendImageData();

	(* <ProductionSite> tag *)
	strString := F_CONCAT4(strPrefix, '$T$T<ProductionSite>', stOACData.OuterMachine.ProductionSite, '</ProductionSite>$R$N');
	AppendImageData();

	(* <ProductionLine> tag *)
	strString := F_CONCAT4(strPrefix, '$T$T<ProductionLine>', stOACData.OuterMachine.ProductionLine, '</ProductionLine>$R$N');
	AppendImageData();

	(* <OuterMachine> closing tag *)
	strString := CONCAT(strPrefix, '$T</OuterMachine>$R$N');
	AppendImageData();

	(* <strAggregationCodes[1]> field *)
	strString := F_CONCAT6(strPrefix, '$T<AggregationCodes index="','1', '"><![CDATA[',stOACData.AggregationCodes[1], ']]></AggregationCodes>$R$N');
	AppendImageData();

	(* <strAggregationCodes[2]> field *)
	strString := F_CONCAT6(strPrefix, '$T<AggregationCodes index="', '2', '"><![CDATA[',stOACData.AggregationCodes[2], ']]></AggregationCodes>$R$N');
	AppendImageData();

	(* <OuterMasterListRestored> field *)
	strString := F_CONCAT4(strPrefix, '$T<OuterMasterListRestored>', BOOL_TO_STRING(stOACData.OuterMasterListRestored), '</OuterMasterListRestored>$R$N');
	AppendImageData();

	(* <CodingAndTrackingMode> field *)
	strString := F_CONCAT4(strPrefix, '$T<CodingAndTrackingMode>', INT_TO_STRING(stOACData.CodingAndTrackingMode), '</CodingAndTrackingMode>$R$N');
	AppendImageData();

	(* <NumberOfPacks> field *)
	strString := F_CONCAT4(strPrefix, '$T<NumberOfPacks>', INT_TO_STRING(stOACData.NumberOfPacks), '</NumberOfPacks>$R$N');
	AppendImageData();

	(* <AcceptanceLevel> field *)
	strString := F_CONCAT4(strPrefix, '$T<AcceptanceLevel>', INT_TO_STRING(stOACData.AcceptanceLevel), '</AcceptanceLevel>$R$N');
	AppendImageData();

	(* <NumberOfLinkedPacks> field *)
	strString := F_CONCAT4(strPrefix, '$T<NumberOfLinkedPacks>', INT_TO_STRING(stOACData.NumberOfLinkedPacks), '</NumberOfLinkedPacks>$R$N');
	AppendImageData();

	(* <BatchNumber> field *)
	strString := F_CONCAT4(strPrefix, '$T<BatchNumber>', stOACData.BatchNumber, '</BatchNumber>$R$N');
	AppendImageData();

	(* <DataSource> field *)
	strString := F_CONCAT4(strPrefix, '$T<DataSource>', stOACData.DataSource, '</DataSource>$R$N');
	AppendImageData();

	(* <OuterRejectCode> field *)
	strString := F_CONCAT4(strPrefix, '$T<OuterRejectCode>', stOACData.OuterRejectCode, '</OuterRejectCode>$R$N');
	AppendImageData();

	(* <OuterRejectID> field *)
	strString := F_CONCAT4(strPrefix, '$T<OuterRejectID>', UINT_TO_STRING(stOACData.OuterRejectID), '</OuterRejectID>$R$N');
	AppendImageData();

	(* <OuterCodeStatus> field *)
	strString := F_CONCAT4(strPrefix, '$T<OuterCodeStatus>', WORD_TO_STRING(stOACData.OuterCodeStatus), '</OuterCodeStatus>$R$N');
	AppendImageData();

	(* max number of Packs/Outer *)
	nMaxPackIndex := UDINT_TO_INT(SIZEOF(stOACData.PackCode) / SIZEOF(stOACData.PackCode[1]));

	(* OAC data contains pack codes number of packs is valid *)
	IF stOACData.NumberOfPacks > 0 AND stOACData.NumberOfPacks <= nMaxPackIndex THEN

		(* for each pack code *)
		FOR nPackIndex := 1 TO stOACData.NumberOfPacks DO

			(* <PackCode index="xx"> field *)
			strString := F_CONCAT6(strPrefix, '$T<PackCode index="', INT_TO_STRING(nPackIndex), '"><![CDATA[', stOACData.PackCode[nPackIndex], ']]></PackCode>$R$N');
			AppendImageData();
		END_FOR

	(* for each pack code *)
		FOR nPackIndex := 1 TO stOACData.NumberOfPacks DO

			(* <PackRejectCode index="xx"> field *)
			strString := F_CONCAT6(strPrefix, '$T<PackRejectCode index="', INT_TO_STRING(nPackIndex), '">', stOACData.PackRejectCode[nPackIndex], '</PackRejectCode>$R$N');
			AppendImageData();
		END_FOR

	(* for each pack code *)
		FOR nPackIndex := 1 TO stOACData.NumberOfPacks DO

			(* <PackRejectID index="xx"> field *)
			strString := F_CONCAT6(strPrefix, '$T<PackRejectID index="', INT_TO_STRING(nPackIndex), '">', UINT_TO_STRING(stOACData.PackRejectID[nPackIndex]), '</PackRejectID>$R$N');
			AppendImageData();
		END_FOR

		(* for each pack code *)
		FOR nPackIndex := 1 TO stOACData.NumberOfPacks DO
			(* <PackCodeStatus index="xx"> field *)
			strString := F_CONCAT6(strPrefix, '$T<PackCodeStatus index="', INT_TO_STRING(nPackIndex), '">', WORD_TO_STRING(stOACData.PackCodeStatus[nPackIndex]), '</PackCodeStatus>$R$N');
			AppendImageData();
		END_FOR

	END_IF

	(* <Outer> closing tag *)
	strString := CONCAT(strPrefix, '</Outer>$R$N');
	AppendImageData();

	(* update outputs *)
	bDone := TRUE;

(* unknown state *)
ELSIF bExecute = FALSE THEN

	(* clear outputs *)
	bDone := FALSE;
END_IF

ACTION AppendImageData:
nStringLen := LEN(strString);
nControlSize := nControlSize + nStringLen;
IF nControlSize <  nMaxOACImageSize THEN
	MEMMOVE(ADR(arrOACImage[nOACByte]), ADR(strString), nStringLen);
	nOACByte := nOACByte + nStringLen;
ELSE
	bBufferOverflow	:=TRUE;
	bDone := TRUE;
	(*RETURN;*)
END_IF
END_ACTION

END_FUNCTION_BLOCK

// ---- POUs/_Exclude/OCV FBs/FB_OCV_WriteFile.TcPOU
FUNCTION_BLOCK FB_OCV_WriteFile
VAR_INPUT
	bExecute					: BOOL;			(* scan for valid Outer in arrOuterStatus *)
	sTargetPath				: STRING(255);	(* target folder for OCV file *)
	ePackAggregationMode	: E_SYSTEM_PackAggregationMode ;
	nPacksPerOuter			: INT;
	aOCVFileCodeName		: ARRAY[1..2] OF T_MaxString;
	bSkipWriteFile1			: BOOL;
	bSkipWriteFile2			: BOOL;
	stOCVPackStatus			: ST_OUTER_Status;	(*  OCV queue status *)
END_VAR
VAR_OUTPUT
	bDone						: BOOL;			(* TRUE = write OCV file complete *)
	bBusy						: BOOL;			(* TRUE = write OCV file in progress *)
	bError						: BOOL;			(* TRUE = write OCV file error *)
	nErrorID					: UDINT;		(* error ID *)
	sOCVFile1					: T_OCV_Filename;	(* OCV file name *)
	sOCVFile2					: T_OCV_Filename;	(* OCV file name *)
	nStoredFiles				: INT;
END_VAR
VAR
	fbExecute					: R_TRIG;
	eState						: E_OUTER_State;
	eErrorState					: E_OUTER_State;
	fbBuildOCVData			: FB_OCV_BuildXMLData;
	fbCreateFolder				: FB_CreateDir;
	fbWriteFile					: FB_FILE_WriteByByte;
	sOCVTempName			: T_OCV_Filename;

END_VAR

(* monitor bExecute for rising edge *)
fbExecute(CLK := bExecute);

CASE eState OF

	(* idle *)
	E_OUTER_IDLE:

		(* rising edge on bExecute *)
		IF fbExecute.Q = TRUE THEN

			(* update outputs *)
			bDone := FALSE;
			bBusy := TRUE;
			bError := FALSE;
			nErrorID := 0;
			nStoredFiles := 0;
			sOCVFile1 := '';
			sOCVFile2 :='';

			eState := E_OUTER_BUILDXMLIMAGE;

		(* disabled *)
		ELSIF bExecute = FALSE THEN

			(* update outputs *)
			bDone := FALSE;
			bBusy := FALSE;
			(*bError := FALSE;
			nErrorID := 0;*)
			nStoredFiles := 0;

		END_IF

	(* build OCV image in XML format *)
	E_OUTER_BUILDXMLIMAGE:

		(* build OAC data *)
		fbBuildOCVData(
			bExecute		:= TRUE,
			bAddXMLHeader	:= TRUE,
			nTabIndent		:= 0,
			nPacksPerOuter 	:= nPacksPerOuter,
			stOCVDataToImage 	:= stOCVPackStatus,
			ePackAggregationMode	:= ePackAggregationMode
		);

		(* build OCV data complete *)
		IF fbBuildOCVData.bDone = TRUE THEN

			eState := E_OUTER_CREATEERRORFOLDER;

			(* close off fbBuild  OCVData *)
			fbBuildOCVData(bExecute := FALSE);
		END_IF

(***************************************************************************)

	(* create folders *)
	E_OUTER_CREATEERRORFOLDER:

		(* create date archive folder *)
		fbCreateFolder(
			sNetId		:= '',
			sPathName	:= sTargetPath,
			ePath		:= PATH_GENERIC,
			bExecute	:= TRUE,
			tTimeout	:= T#300ms
		);

		(* create folder complete *)
		IF fbCreateFolder.bBusy = FALSE THEN

			(* create folder completed OK or folder already exists *)
			IF fbCreateFolder.bError = FALSE OR (fbCreateFolder.bError = TRUE AND fbCreateFolder.nErrId = 16#70C) THEN

				eState := E_OUTER_WRITEXMLIMAGE;
			(* create folder error *)
			ELSE

				(* update outputs *)
				bError := TRUE;
				nErrorID := fbCreateFolder.nErrId;
				eErrorState := eState;

				eState := E_OUTER_DONE;
			END_IF

			(* close off fbCreateFolder *)
			fbCreateFolder(bExecute := FALSE);
		END_IF

(***************************************************************************)

	(* write OCV image to file *)
	E_OUTER_WRITEXMLIMAGE:

		IF NOT bSkipWriteFile1 THEN
			(* write XML template to file *)

			sOCVFile1 := F_CONCAT3('OCV_', aOCVFileCodeName[1], '.xml');

			fbWriteFile(
				bExecute	:= TRUE,
				pSourceAddr	:= ADR(fbBuildOCVData.arrOCVImage),
				nSourceSize	:= fbBuildOCVData.nOCVByte,
				strPathFile	:= CONCAT(sTargetPath,sOCVFile1),
				tTimeout	:= cHALF_SECOND
			);

			(* file write complete *)
			IF fbWriteFile.bDone = TRUE THEN
				sOCVTempName	:= sOCVFile1;
				(* file write completed OK *)
				IF fbWriteFile.bError = FALSE THEN

					nStoredFiles := nStoredFiles +1;
	
				(* file write error *)
				ELSE
	
					bError := TRUE;
					nErrorID := fbWriteFile.nErrorID;
					eErrorState := eState;
				END_IF
	
				eState := E_OUTER_WRITESECONDXMLIMAGE;
	
				(* close of fbWriteFile *)
				fbWriteFile(bExecute := FALSE);
			END_IF
		ELSE
			eState := E_OUTER_WRITESECONDXMLIMAGE;
		END_IF

	E_OUTER_WRITESECONDXMLIMAGE:

	IF NOT bSkipWriteFile2 THEN
	(* write XML template to file *)

		sOCVFile2 := F_CONCAT3('OCV_', aOCVFileCodeName[2], '.xml');

		fbWriteFile(
			bExecute	:= TRUE,
			pSourceAddr	:= ADR(fbBuildOCVData.arrOCVImage),
			nSourceSize	:= fbBuildOCVData.nOCVByte,
			strPathFile	:=  CONCAT(sTargetPath, sOCVFile2),
			tTimeout	:= cHALF_SECOND
		);

		(* file write complete *)
		IF fbWriteFile.bDone = TRUE THEN
			sOCVTempName	:= sOCVFile2;
			(* file write completed OK *)
			IF fbWriteFile.bError = FALSE THEN

				nStoredFiles := nStoredFiles +1;

			(* file write error *)
			ELSE

				bError := TRUE;
				nErrorID := fbWriteFile.nErrorID;
				eErrorState := eState;
			END_IF

			eState := E_OUTER_DONE;

			(* close of fbWriteFile *)
			fbWriteFile(bExecute := FALSE);
		END_IF
	ELSE
		eState := E_OUTER_DONE;
	END_IF

	(* OCV file complete *)
	E_OUTER_DONE:

		(* update outputs *)
		bDone := TRUE;
		bBusy := FALSE;

		eState := E_OUTER_IDLE;


(* unknown state *)
ELSE

	eState := E_OUTER_IDLE;
END_CASE

END_FUNCTION_BLOCK

// ---- POUs/_Exclude/OCV FBs/FB_OCV_BuildXMLData.TcPOU
FUNCTION_BLOCK FB_OCV_BuildXMLData
VAR_INPUT
	bExecute					: BOOL;
	bAddXMLHeader			: BOOL;
	nTabIndent					: BYTE;
	nPacksPerOuter			: INT;
	stOCVDataToImage		: ST_OUTER_Status;	(*  OCV queue status *)
	ePackAggregationMode	: E_SYSTEM_PackAggregationMode ;
END_VAR
VAR_OUTPUT
	bDone					: BOOL;
	nOCVByte					: INT;		(* total bytes for OCV template *)
	arrOCVImage				: ARRAY[0..20000] OF BYTE;
	bBufferOverflow			: BOOL;
END_VAR
VAR
	fbExecute					: R_TRIG;
	strPrefix					: T_MaxString; (*STRING(1); fixes write issue*)
	strString					: STRING(255);
	nStringLen				: INT;
	nMaxOCVImageSize			: UINT;
	nControlSize				: UINT;
	nMaxPackIndex			: INT;
	nPackIndex				: INT;
	(*nChecksum				: WORD;*)
END_VAR

(* rising edge of bExecute *)
fbExecute(CLK := bExecute);

(* rising edge of bExecute *)
IF fbExecute.Q = TRUE THEN

	(* update outputs *)
	bDone := FALSE;
	bBufferOverflow	:=FALSE;

	(* clear output array and reset byte counter *)
	MEMSET(ADR(arrOCVImage), 16#00, SIZEOF(arrOCVImage));
	nOCVByte := 0;
	nControlSize := 0;
	nMaxOCVImageSize := SIZEOF(arrOCVImage);

	(* XML header required *)
	IF bAddXMLHeader = TRUE THEN

		(* no prefix required, include XML header *)
		strString := cXML_HEADER;
		nStringLen := LEN(strString);
		MEMMOVE(ADR(arrOCVImage[nOCVByte]), ADR(strString), nStringLen);
		nOCVByte := nOCVByte + nStringLen;
		nControlSize :=	nOCVByte;

		(* <Comment> tag *)
		strString := '<!--File OAC builder. Version 2.2.000 Relase 06.09.2022 PTR -->$R$N';
		AppendImageData();
	END_IF

	(* tab indent required *)
	IF nTabIndent > 0 THEN

		(* generate strPrefix with specified number of tabs *)
		strPrefix := F_StringAddPrefix('$T', nTabIndent, '$T');

	(* no tab index required *)
	ELSE

		(* clear strPrefix *)
		strPrefix := '';
	END_IF

	(* <Pack> tag *)
	strString := CONCAT(strPrefix, '<OCVPack>$R$N');
	AppendImageData();


	(* <nTriggerID> field *)
	strString := F_CONCAT4(strPrefix, '$T<nTriggerID>', UDINT_TO_STRING(stOCVDataToImage.nTriggerID), '</nTriggerID>$R$N');
	AppendImageData();


	(* <strDataSourceTracker> field *)
	strString := F_CONCAT4(strPrefix, '$T<sDataSourceTracker>', stOCVDataToImage.sDataSourceTracker, '</sDataSourceTracker>$R$N');
	AppendImageData();


	(* <stOACData> field *)
	strString := CONCAT(strPrefix, '$T<stOACData>$R$N');
	AppendImageData();


	(* <ProductionDate> field *)
	strString := F_CONCAT4(strPrefix, '$T$T<ProductionDate>', stOCVDataToImage.stOACData.ProductionDate, '</ProductionDate>$R$N');
	AppendImageData();


	(* <ProductionTime> field *)
	strString := F_CONCAT4(strPrefix, '$T$T<ProductionTime>', stOCVDataToImage.stOACData.ProductionTime, '</ProductionTime>$R$N');
	AppendImageData();


	(* <ProductionTimeOffset> field *)
	strString := F_CONCAT4(strPrefix, '$T$T<ProductionTimeOffset>', stOCVDataToImage.stOACData.ProductionTimeOffset, '</ProductionTimeOffset>$R$N');
	AppendImageData();


	(* <PackTimeStamp> field *)
	strString := F_CONCAT4(strPrefix, '$T$T<PackTimeStamp>', stOCVDataToImage.stOACData.PackTimeStamp, '</PackTimeStamp>$R$N');
	AppendImageData();


	(* <strAggregationCodes[1]> field *)
	strString := F_CONCAT6(strPrefix, '$T$T<AggregationCodes index="','1', '"><![CDATA[',stOCVDataToImage.stOACData.AggregationCodes[1], ']]></AggregationCodes>$R$N');
	AppendImageData();


	(* <strAggregationCodes[2]> field *)
	strString := F_CONCAT6(strPrefix, '$T$T<AggregationCodes index="', '2', '"><![CDATA[',stOCVDataToImage.stOACData.AggregationCodes[2], ']]></AggregationCodes>$R$N');
	AppendImageData();


	(* <CodingAndTrackingMode> field *)
	strString := F_CONCAT4(strPrefix, '$T$T<CodingAndTrackingMode>', INT_TO_STRING(stOCVDataToImage.stOACData.CodingAndTrackingMode), '</CodingAndTrackingMode>$R$N');
	AppendImageData();


	(* <NumberOfPacks> field *)
	strString := F_CONCAT4(strPrefix, '$T$T<NumberOfPacks>', INT_TO_STRING(stOCVDataToImage.stOACData.NumberOfPacks), '</NumberOfPacks>$R$N');
	AppendImageData();


	(* <AcceptanceLevel> field *)
	strString := F_CONCAT4(strPrefix, '$T$T<AcceptanceLevel>', INT_TO_STRING(stOCVDataToImage.stOACData.AcceptanceLevel), '</AcceptanceLevel>$R$N');
	AppendImageData();


	(* <NumberOfLinkedPacks> field *)
	strString := F_CONCAT4(strPrefix, '$T$T<NumberOfLinkedPacks>', INT_TO_STRING(stOCVDataToImage.stOACData.NumberOfLinkedPacks), '</NumberOfLinkedPacks>$R$N');
	AppendImageData();


	(* max number of Packs*)
	nMaxPackIndex := UDINT_TO_INT(SIZEOF(stOCVDataToImage.stOACData.PackCode) / SIZEOF(stOCVDataToImage.stOACData.PackCode[1]));

	(* OCV data contains pack codes number of packs is valid *)
	IF nPacksPerOuter > 0 AND nPacksPerOuter <= nMaxPackIndex THEN

		(* for each pack code *)
		FOR nPackIndex := 1 TO nPacksPerOuter DO
			(* <PackCode index="xx"> field *)
			strString := F_CONCAT6(strPrefix, '$T$T<PackCode index="', INT_TO_STRING(nPackIndex), '"><![CDATA[', stOCVDataToImage.stOACData.PackCode[nPackIndex], ']]></PackCode>$R$N');
			AppendImageData();
		END_FOR

		(* for each pack code *)
		FOR nPackIndex := 1 TO nPacksPerOuter DO
			(* <PackRejectCode index="xx"> field *)
			strString := F_CONCAT6(strPrefix, '$T$T<PackRejectCode index="', INT_TO_STRING(nPackIndex), '">', stOCVDataToImage.stOACData.PackRejectCode[nPackIndex], '</PackRejectCode>$R$N');
			AppendImageData();
		END_FOR

		(* for each pack code *)
		FOR nPackIndex := 1 TO nPacksPerOuter DO
			(* <PackRejectID index="xx"> field *)
			strString := F_CONCAT6(strPrefix, '$T$T<PackRejectID index="', INT_TO_STRING(nPackIndex), '">', UINT_TO_STRING(stOCVDataToImage.stOACData.PackRejectID[nPackIndex]), '</PackRejectID>$R$N');
			AppendImageData();
		END_FOR

		(* for each pack code *)
		FOR nPackIndex := 1 TO nPacksPerOuter DO
			(* <PackCodeStatus index="xx"> field *)
			strString := F_CONCAT6(strPrefix, '$T$T<PackCodeStatus index="', INT_TO_STRING(nPackIndex), '">', WORD_TO_STRING(stOCVDataToImage.stOACData.PackCodeStatus[nPackIndex]), '</PackCodeStatus>$R$N');
			AppendImageData();
		END_FOR
	END_IF

	(* <Outer> closing tag *)
	strString := CONCAT(strPrefix, '$T</stOACData>$R$N');
	AppendImageData();


	(* OCV data contains pack codes number of packs is valid *)
	IF nPacksPerOuter > 0 AND nPacksPerOuter <= nMaxPackIndex THEN

		(* for each pack code *)
		FOR nPackIndex := 1 TO nPacksPerOuter DO

		(* <stOCVDataToImage.aOACPackStatus index="xx"> field *)
			strString := F_CONCAT6(strPrefix, '$T<aOACPackStatus index="', INT_TO_STRING(nPackIndex), '">',BYTE_TO_STRING(stOCVDataToImage.aOACPackStatus[nPackIndex]), '</aOACPackStatus>$R$N');
			AppendImageData();
		END_FOR

	(* for each pack code *)
		(*FOR nPackIndex := 1 TO nPacksPerOuter DO

		(* <stOCVDataToImage.aOACPackStatus index="xx"> field *)
			strString := F_CONCAT6(strPrefix, '$T<aPackSUPIResult index="', INT_TO_STRING(nPackIndex), '">',DINT_TO_STRING(stOCVDataToImage.aPackSUPIResult[nPackIndex]), '</aPackSUPIResult>$R$N');
			AppendImageData();
		END_FOR*)

	END_IF

	CASE ePackAggregationMode OF

	E_SYSTEM_PAOL_2CAM, E_SYSTEM_PAOL_3CAM:

		IF nPacksPerOuter > 0 AND nPacksPerOuter <= nMaxPackIndex THEN

			(* for each pack code *)
			FOR nPackIndex := 1 TO nPacksPerOuter DO

			(* <sPackCodes index="xx"> field *)
				strString := F_CONCAT4(strPrefix, '$T<sPackCodes index="', INT_TO_STRING(nPackIndex), '">$R$N');
				AppendImageData();


				(* <sBuffer index="1"> field *)
				strString := CONCAT(strPrefix, '$T$T<sBuffer index="1">$R$N');
				AppendImageData();


				(* <strCode> field *)
				strString := F_CONCAT4(strPrefix, '$T$T$T<strCode><![CDATA[', stOCVDataToImage.aPackCodes[nPackIndex].sBuffer[1].strCode  , ']]></strCode>$R$N');
				AppendImageData();


				(* <nStringSize> field *)
				strString := F_CONCAT4(strPrefix, '$T$T$T<nStringSize>', INT_TO_STRING(stOCVDataToImage.aPackCodes[nPackIndex].sBuffer[1].nStringSize)  , '</nStringSize>$R$N');
				AppendImageData();


				(* <nStringSize> field *)
				strString := F_CONCAT4(strPrefix, '$T$T$T<nStatus>', BYTE_TO_STRING(stOCVDataToImage.aPackCodes[nPackIndex].sBuffer[1].nStatus)  , '</nStatus>$R$N');
				AppendImageData();


				(* close <sBuffer index="1"> field *)
				strString := CONCAT(strPrefix, '$T$T</sBuffer>$R$N');
				AppendImageData();


				(* <sBuffer index="2"> field *)
				strString := CONCAT(strPrefix, '$T$T<sBuffer index="2">$R$N');
				AppendImageData();

	
				(* <strCode> field *)
				strString := F_CONCAT4(strPrefix, '$T$T$T<strCode><![CDATA[', stOCVDataToImage.aPackCodes[nPackIndex].sBuffer[2].strCode  , ']]></strCode>$R$N');
				AppendImageData();


				(* <nStringSize> field *)
				strString := F_CONCAT4(strPrefix, '$T$T$T<nStringSize>', INT_TO_STRING(stOCVDataToImage.aPackCodes[nPackIndex].sBuffer[2].nStringSize)  , '</nStringSize>$R$N');
				AppendImageData();


				(* <nStringSize> field *)
				strString := F_CONCAT4(strPrefix, '$T$T$T<nStatus>', BYTE_TO_STRING(stOCVDataToImage.aPackCodes[nPackIndex].sBuffer[2].nStatus)  , '</nStatus>$R$N');
				AppendImageData();


				(* close <sBuffer index="2"> field *)
				strString := CONCAT(strPrefix, '$T$T</sBuffer>$R$N');
				AppendImageData();


				(* <sPackCodes index="xx"> field *)
				strString := CONCAT(strPrefix, '$T</sPackCodes>$R$N');
				AppendImageData();


			END_FOR
		END_IF

	E_SYSTEM_PLAS_T01:

		(* FOR each pack code *)(* OCV data contains pack codes number of packs is valid *)
		IF nPacksPerOuter > 0 AND nPacksPerOuter <= nMaxPackIndex THEN
	
			(* for each pack code *)
			FOR nPackIndex := 1 TO nPacksPerOuter DO

			(* <stOCVDataToImage.aPackCodeFilledIn index="xx"> field *)
				strString := F_CONCAT6(strPrefix, '$T<aPackCodeFilledIn index="', INT_TO_STRING(nPackIndex), '">',INT_TO_STRING(stOCVDataToImage.aPackCodeFilledIn[nPackIndex]), '</aPackCodeFilledIn>$R$N');
				AppendImageData();
			END_FOR
		END_IF

	E_SYSTEM_PLAS_T02, E_SYSTEM_PLAS_T03, E_SYSTEM_PLAS_T04:

		(* FOR each pack code *)(* OCV data contains pack codes number of packs is valid *)
		IF nPacksPerOuter > 0 AND nPacksPerOuter <= nMaxPackIndex THEN

			(* for each pack code *)
			FOR nPackIndex := 1 TO nPacksPerOuter DO

			(* <stOCVDataToImage.aPackCodeFilledIn index="xx"> field *)
				strString := F_CONCAT6(strPrefix, '$T<aPackCodeFilledIn index="', INT_TO_STRING(nPackIndex), '">',INT_TO_STRING(stOCVDataToImage.aPackCodeFilledIn[nPackIndex]), '</aPackCodeFilledIn>$R$N');
				AppendImageData();
			END_FOR
		END_IF

	END_CASE

	(* <Outer> closing tag *)
	strString := CONCAT(strPrefix, '</OCVPack>$R$N');
	AppendImageData();

	(* update outputs *)
	bDone := TRUE;

(* unknown state *)
ELSIF bExecute = FALSE THEN

	(* clear outputs *)
	bDone := FALSE;
END_IF

ACTION AppendImageData:
nStringLen := LEN(strString);
nControlSize := nControlSize + nStringLen;
IF nControlSize <  nMaxOCVImageSize THEN
	MEMMOVE(ADR(arrOCVImage[nOCVByte]), ADR(strString), nStringLen);
	nOCVByte := nOCVByte + nStringLen;
ELSE
	bBufferOverflow	:=TRUE;
	bDone := TRUE;
	(*RETURN;*)
END_IF
END_ACTION

END_FUNCTION_BLOCK

// ---- POUs/_Exclude/C09_MaintainFolders_ORG.TcPOU
(* delete old files and delete oldest files if number of files exceeds specified number *)
PROGRAM C09_MaintainFolders_ORG
VAR
	tArchiveCheck				: TIME := t#4s;
	fbMaintainArchive			: FB_PulseGenerator;
	tDeleteTimeCheck			: TIME := t#20m;
	fbMaintainDeleteTime		: FB_PulseGenerator;
	(*tDeleteItemCheck			: TIME := t#4s;
	fbMaintainDeleteItem		: FB_PulseGenerator;*)
	nActivateBitWord			: DWORD; (* if index increase 32 bits it is necceasry to declar 64 bits var like LREAL;*)

	fbMaintainFolders			: ARRAY[1..25] OF NT_StartProcess;
	bTest	: BOOL;
	(*fbMoveOHMToArchive		: FB_OHM_MoveToArchive;*)
	(*fbMoveCACToArchive		: FB_CAC_MoveToArchive;*)
	fbMoveCHMToArchive		: FB_CHM_MoveToArchive;
	bZipCHMArchive			: BOOL;
	rtrigZipAfetrPassthrough		: R_TRIG;
	bManualZip					: BOOL;

	(*fbCompresOHMArchive		: NT_StartProcess;
	fbCompresCHMArchive		: NT_StartProcess;
	fbCompresPHMArchive		: NT_StartProcess;

	fbDeleteCHMNoLabel		: NT_StartProcess;*)

	fbRestoreTimer			: TON;
	fbRestoreOACFromCAC		: FB_CAC_RestoreOAC;
	nOCVFilesRestored			: UDINT;
	nOACFilesRestored			: UDINT;
	nCACFilesRestored			: UDINT;

	(*rtrigClearOCV				: R_TRIG;
	rtrigClearOCVError			: R_TRIG;
	rtrigClearOAC				: R_TRIG;
	rtrigClearOACError			: R_TRIG;

	fbClearOCVArchive			: FB_OCV_ClearArchive;
	fbClearOCVError			: FB_OCV_ClearArchive;
	fbClearOACArchive			: FB_OAC_ClearArchive;
	fbClearOACError			: FB_OAC_ClearArchive;

	rtrigClearOHM_FLG			: R_TRIG;
	rtrigClearCHM_FLG			: R_TRIG;

	fbClearOHM_FLG			: FB_OHM_ClearFLG;
	fbClearCHM_FLG			: FB_CHM_ClearFLG;
	btest : BOOL;*)

(********************************************************************************
		cBASE_FOLDER_ARR	: ARRAY[1..cSYSTEM_FOLDER_LIMIT] OF T_FolderName :=
			(*01*)'Bridge\',		(*02*)'Bridge\Archive\',		(*03*)'Bridge\Restore\',
			(*04*)'CAC\',		(*05*)'CAC\Archive\',		(*06*)'CAC\Error\',		(*07*)'CAC\Restore\', 	(*08*)'CAC\Restore\Archive\',
			(*09*)'CHM\',		(*10*)'CHM\Archive\',		(*11*)'CHM\Error\',		(*12*)'CHM\OK\',		(*13*)'CHM\Commissioning_Mode\',
			(*14*)'HMI\',
			(*15*)'KPI\',		(*16*)'KPI\Archive\',			(*17*)'KPI\Shift\',		(*18*)'KPI\ProdOrder\',
			(*19*)'OAC\',		(*20*)'OAC\Error\',
			(*21*)'OCV\',		(*22*)'OCV\Error\',
			(*23*)'OHM\',		(*24*)'OHM\Archive\',		(*25*)'OHM\Error\',		(*26*)'OHM\OK\',		(*27*)'OHM\Pending\',
			(*28*)'PCM\',		(*29*)'PCM\Archive\',		(*30*)'PCM\Error\',		(*31*)'PCM\Incoming\',
			(*32*)'PAC\',
			(*33*)'PHM\',		(*34*)'PHM\Archive\',		(*35*)'PHM\Error\',		(*36*)'PHM\OK\',
			(*37*)'Settings\',	(*38*)'Settings\Backups\',
			(*39*)'Templates\',
			(*40*)'Orca\',
			(*41*) 'SystemLog\';

*************************************************************************************)
END_VAR

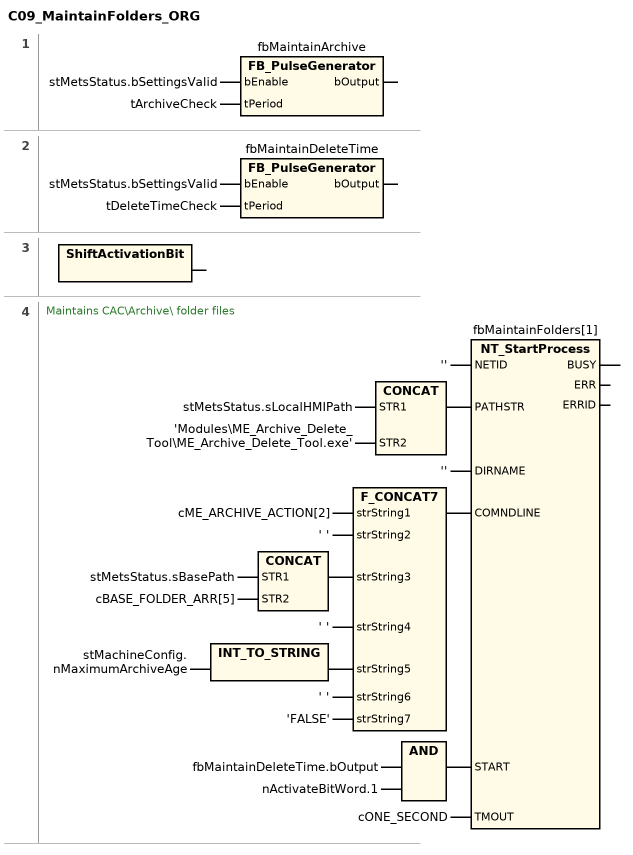
// NETWORK 1
fbMaintainArchive(bEnable := stMetsStatus.bSettingsValid, tPeriod := tArchiveCheck); // FB_PulseGenerator

// NETWORK 2
fbMaintainDeleteTime(bEnable := stMetsStatus.bSettingsValid, tPeriod := tDeleteTimeCheck); // FB_PulseGenerator

// NETWORK 3
ShiftActivationBit();

// NETWORK 4
// Maintains CAC\Archive\ folder files
fbMaintainFolders[1](
    NETID := '',
    PATHSTR := CONCAT(STR1 := stMetsStatus.sLocalHMIPath, STR2 := 'Modules\ME_Archive_Delete_Tool\ME_Archive_Delete_Tool.exe'),
    DIRNAME := '',
    COMNDLINE := F_CONCAT7(strString1 := cME_ARCHIVE_ACTION[2], strString2 := ' ', strString3 := CONCAT(STR1 := stMetsStatus.sBasePath, STR2 := cBASE_FOLDER_ARR[5]), strString4 := ' ', strString5 := INT_TO_STRING(stMachineConfig.nMaximumArchiveAge), strString6 := ' ', strString7 := 'FALSE'),
    START := fbMaintainDeleteTime.bOutput AND nActivateBitWord.1,
    TMOUT := cONE_SECOND); // NT_StartProcess

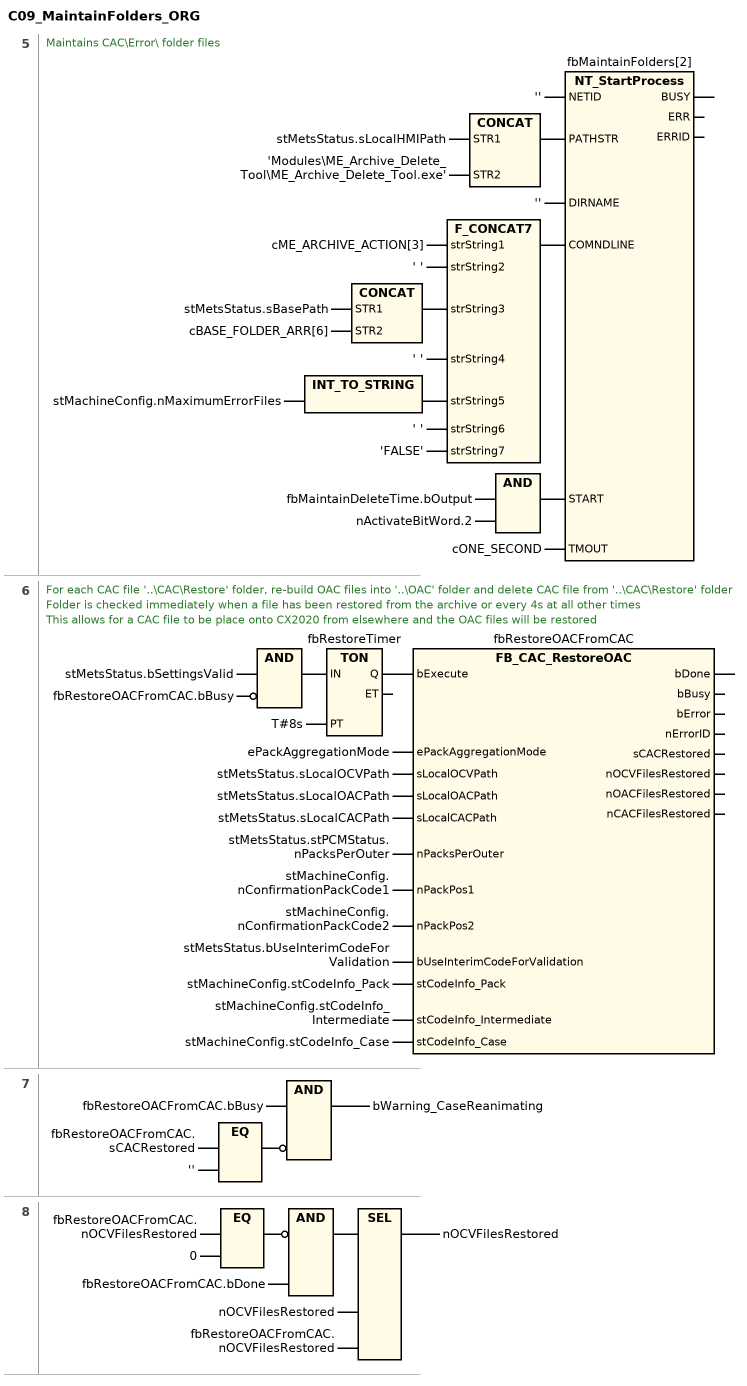
// NETWORK 5
// Maintains CAC\Error\ folder files
fbMaintainFolders[2](
    NETID := '',
    PATHSTR := CONCAT(STR1 := stMetsStatus.sLocalHMIPath, STR2 := 'Modules\ME_Archive_Delete_Tool\ME_Archive_Delete_Tool.exe'),
    DIRNAME := '',
    COMNDLINE := F_CONCAT7(strString1 := cME_ARCHIVE_ACTION[3], strString2 := ' ', strString3 := CONCAT(STR1 := stMetsStatus.sBasePath, STR2 := cBASE_FOLDER_ARR[6]), strString4 := ' ', strString5 := INT_TO_STRING(stMachineConfig.nMaximumErrorFiles), strString6 := ' ', strString7 := 'FALSE'),
    START := fbMaintainDeleteTime.bOutput AND nActivateBitWord.2,
    TMOUT := cONE_SECOND); // NT_StartProcess

// NETWORK 6
// 					For each CAC file '..\CAC\Restore' folder, re-build OAC files into '..\OAC' folder and delete CAC file from '..\CAC\Restore' folder
// Folder is checked immediately when a file has been restored from the archive or every 4s at all other times
// This allows for a CAC file to be place onto CX2020 from elsewhere and the OAC files will be restored
//
fbRestoreTimer(IN := stMetsStatus.bSettingsValid AND NOT fbRestoreOACFromCAC.bBusy, PT := T#8s); // TON
fbRestoreOACFromCAC(
    bExecute := fbRestoreTimer.Q,
    ePackAggregationMode := ePackAggregationMode,
    sLocalOCVPath := stMetsStatus.sLocalOCVPath,
    sLocalOACPath := stMetsStatus.sLocalOACPath,
    sLocalCACPath := stMetsStatus.sLocalCACPath,
    nPacksPerOuter := stMetsStatus.stPCMStatus.nPacksPerOuter,
    nPackPos1 := stMachineConfig.nConfirmationPackCode1,
    nPackPos2 := stMachineConfig.nConfirmationPackCode2,
    bUseInterimCodeForValidation := stMetsStatus.bUseInterimCodeForValidation,
    stCodeInfo_Pack := stMachineConfig.stCodeInfo_Pack,
    stCodeInfo_Intermediate := stMachineConfig.stCodeInfo_Intermediate,
    stCodeInfo_Case := stMachineConfig.stCodeInfo_Case); // FB_CAC_RestoreOAC

// NETWORK 7
bWarning_CaseReanimating := fbRestoreOACFromCAC.bBusy AND NOT (fbRestoreOACFromCAC.sCACRestored = '');

// NETWORK 8
nOCVFilesRestored := SEL(NOT (fbRestoreOACFromCAC.nOCVFilesRestored = 0) AND fbRestoreOACFromCAC.bDone, nOCVFilesRestored, fbRestoreOACFromCAC.nOCVFilesRestored);

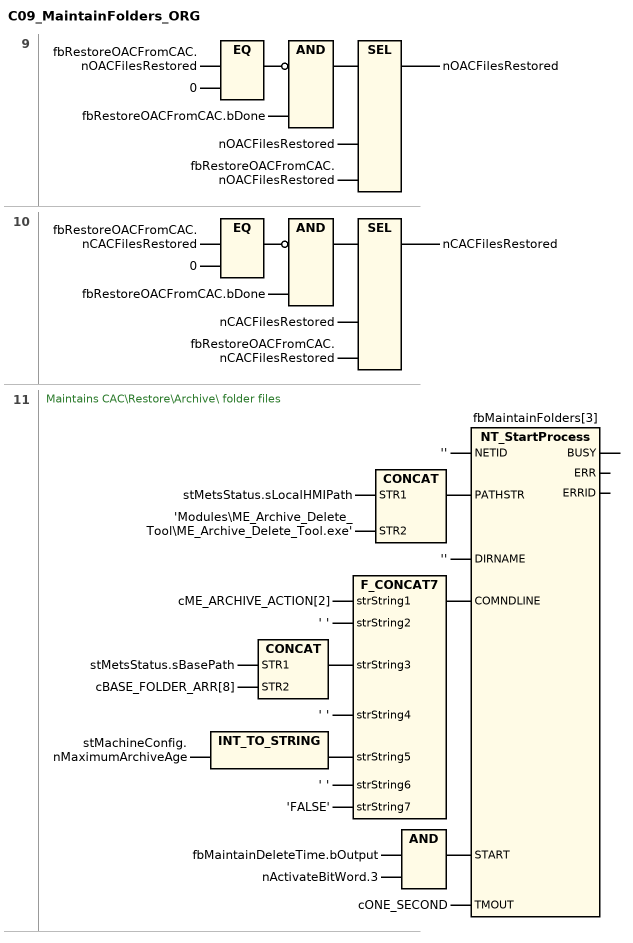
// NETWORK 9
nOACFilesRestored := SEL(NOT (fbRestoreOACFromCAC.nOACFilesRestored = 0) AND fbRestoreOACFromCAC.bDone, nOACFilesRestored, fbRestoreOACFromCAC.nOACFilesRestored);

// NETWORK 10
nCACFilesRestored := SEL(NOT (fbRestoreOACFromCAC.nCACFilesRestored = 0) AND fbRestoreOACFromCAC.bDone, nCACFilesRestored, fbRestoreOACFromCAC.nCACFilesRestored);

// NETWORK 11
// Maintains CAC\Restore\Archive\ folder files
fbMaintainFolders[3](
    NETID := '',
    PATHSTR := CONCAT(STR1 := stMetsStatus.sLocalHMIPath, STR2 := 'Modules\ME_Archive_Delete_Tool\ME_Archive_Delete_Tool.exe'),
    DIRNAME := '',
    COMNDLINE := F_CONCAT7(strString1 := cME_ARCHIVE_ACTION[2], strString2 := ' ', strString3 := CONCAT(STR1 := stMetsStatus.sBasePath, STR2 := cBASE_FOLDER_ARR[8]), strString4 := ' ', strString5 := INT_TO_STRING(stMachineConfig.nMaximumArchiveAge), strString6 := ' ', strString7 := 'FALSE'),
    START := fbMaintainDeleteTime.bOutput AND nActivateBitWord.3,
    TMOUT := cONE_SECOND); // NT_StartProcess

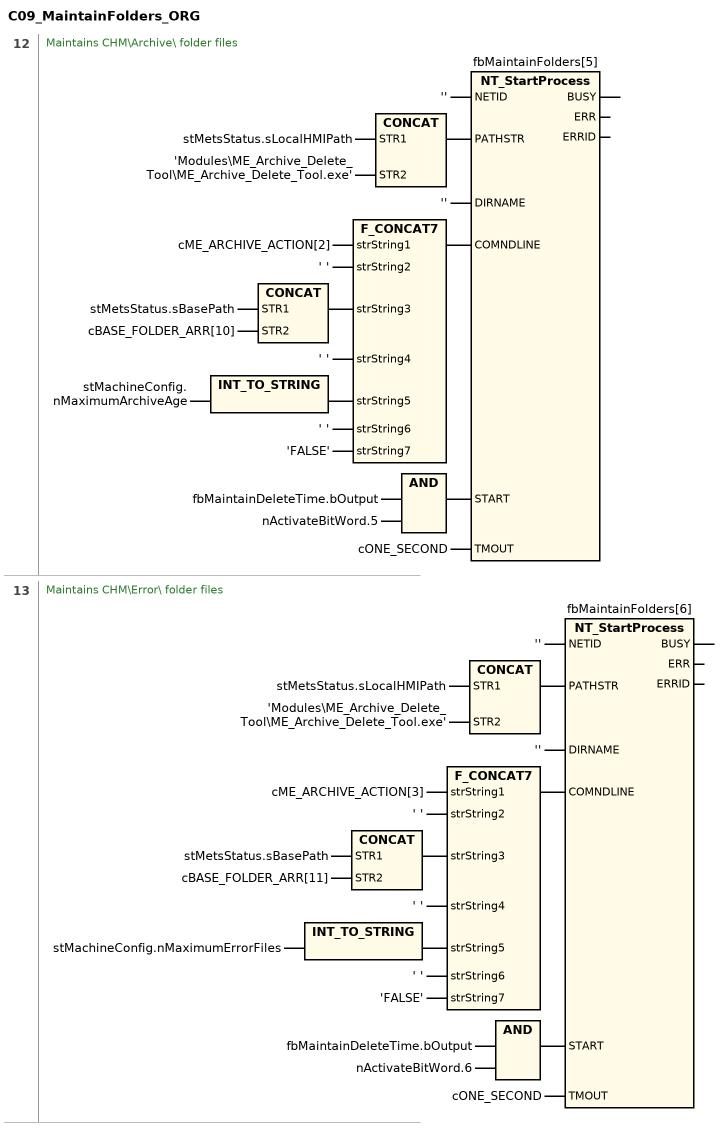
// NETWORK 12
// Maintains CHM\Archive\ folder files
fbMaintainFolders[5](
    NETID := '',
    PATHSTR := CONCAT(STR1 := stMetsStatus.sLocalHMIPath, STR2 := 'Modules\ME_Archive_Delete_Tool\ME_Archive_Delete_Tool.exe'),
    DIRNAME := '',
    COMNDLINE := F_CONCAT7(strString1 := cME_ARCHIVE_ACTION[2], strString2 := ' ', strString3 := CONCAT(STR1 := stMetsStatus.sBasePath, STR2 := cBASE_FOLDER_ARR[10]), strString4 := ' ', strString5 := INT_TO_STRING(stMachineConfig.nMaximumArchiveAge), strString6 := ' ', strString7 := 'FALSE'),
    START := fbMaintainDeleteTime.bOutput AND nActivateBitWord.5,
    TMOUT := cONE_SECOND); // NT_StartProcess

// NETWORK 13
// Maintains CHM\Error\ folder files
fbMaintainFolders[6](
    NETID := '',
    PATHSTR := CONCAT(STR1 := stMetsStatus.sLocalHMIPath, STR2 := 'Modules\ME_Archive_Delete_Tool\ME_Archive_Delete_Tool.exe'),
    DIRNAME := '',
    COMNDLINE := F_CONCAT7(strString1 := cME_ARCHIVE_ACTION[3], strString2 := ' ', strString3 := CONCAT(STR1 := stMetsStatus.sBasePath, STR2 := cBASE_FOLDER_ARR[11]), strString4 := ' ', strString5 := INT_TO_STRING(stMachineConfig.nMaximumErrorFiles), strString6 := ' ', strString7 := 'FALSE'),
    START := fbMaintainDeleteTime.bOutput AND nActivateBitWord.6,
    TMOUT := cONE_SECOND); // NT_StartProcess

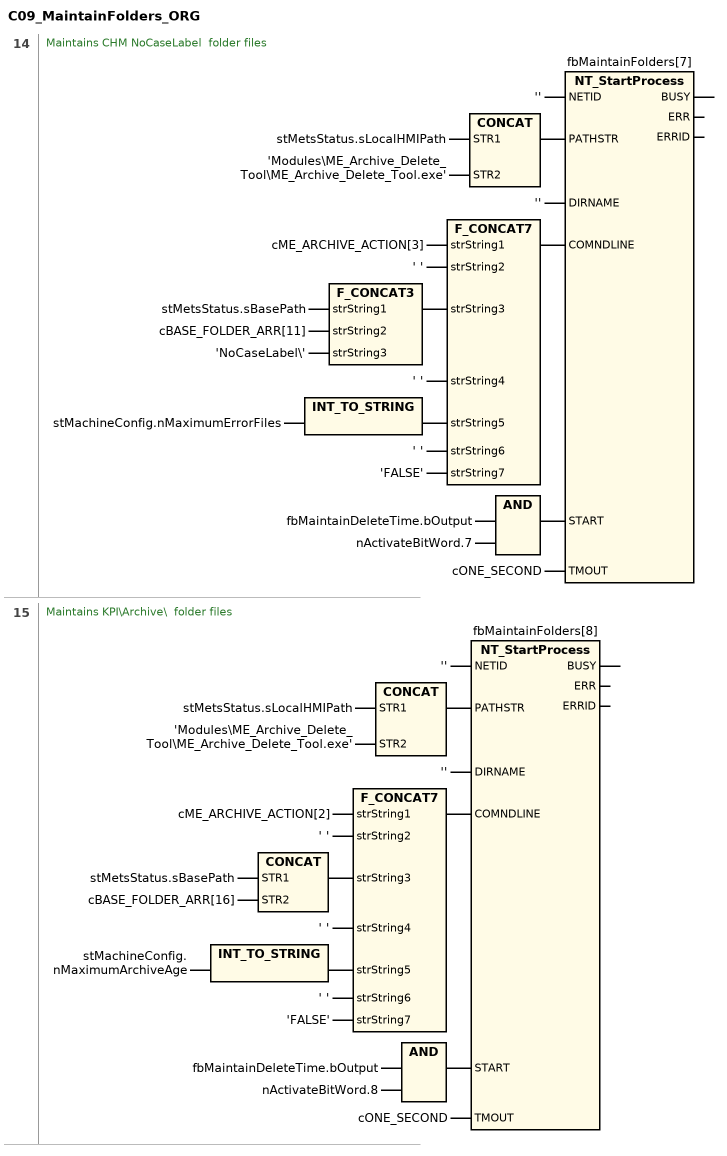
// NETWORK 14
// Maintains CHM NoCaseLabel  folder files
fbMaintainFolders[7](
    NETID := '',
    PATHSTR := CONCAT(STR1 := stMetsStatus.sLocalHMIPath, STR2 := 'Modules\ME_Archive_Delete_Tool\ME_Archive_Delete_Tool.exe'),
    DIRNAME := '',
    COMNDLINE := F_CONCAT7(strString1 := cME_ARCHIVE_ACTION[3], strString2 := ' ', strString3 := F_CONCAT3(strString1 := stMetsStatus.sBasePath, strString2 := cBASE_FOLDER_ARR[11], strString3 := 'NoCaseLabel\'), strString4 := ' ', strString5 := INT_TO_STRING(stMachineConfig.nMaximumErrorFiles), strString6 := ' ', strString7 := 'FALSE'),
    START := fbMaintainDeleteTime.bOutput AND nActivateBitWord.7,
    TMOUT := cONE_SECOND); // NT_StartProcess

// NETWORK 15
// Maintains KPI\Archive\  folder files
fbMaintainFolders[8](
    NETID := '',
    PATHSTR := CONCAT(STR1 := stMetsStatus.sLocalHMIPath, STR2 := 'Modules\ME_Archive_Delete_Tool\ME_Archive_Delete_Tool.exe'),
    DIRNAME := '',
    COMNDLINE := F_CONCAT7(strString1 := cME_ARCHIVE_ACTION[2], strString2 := ' ', strString3 := CONCAT(STR1 := stMetsStatus.sBasePath, STR2 := cBASE_FOLDER_ARR[16]), strString4 := ' ', strString5 := INT_TO_STRING(stMachineConfig.nMaximumArchiveAge), strString6 := ' ', strString7 := 'FALSE'),
    START := fbMaintainDeleteTime.bOutput AND nActivateBitWord.8,
    TMOUT := cONE_SECOND); // NT_StartProcess

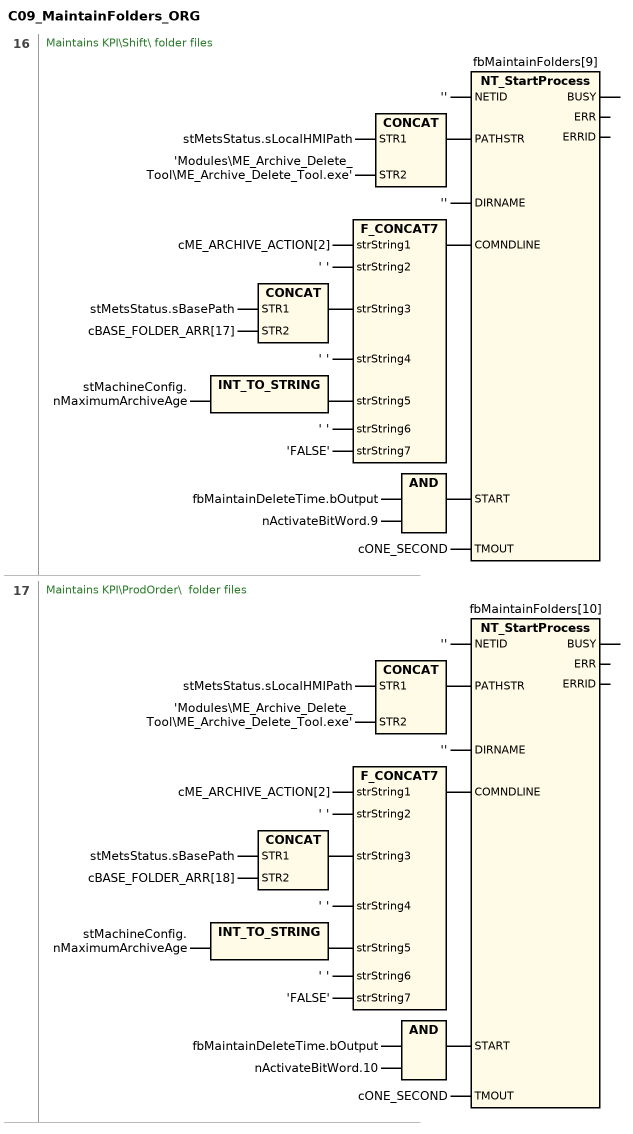
// NETWORK 16
// Maintains KPI\Shift\ folder files
fbMaintainFolders[9](
    NETID := '',
    PATHSTR := CONCAT(STR1 := stMetsStatus.sLocalHMIPath, STR2 := 'Modules\ME_Archive_Delete_Tool\ME_Archive_Delete_Tool.exe'),
    DIRNAME := '',
    COMNDLINE := F_CONCAT7(strString1 := cME_ARCHIVE_ACTION[2], strString2 := ' ', strString3 := CONCAT(STR1 := stMetsStatus.sBasePath, STR2 := cBASE_FOLDER_ARR[17]), strString4 := ' ', strString5 := INT_TO_STRING(stMachineConfig.nMaximumArchiveAge), strString6 := ' ', strString7 := 'FALSE'),
    START := fbMaintainDeleteTime.bOutput AND nActivateBitWord.9,
    TMOUT := cONE_SECOND); // NT_StartProcess

// NETWORK 17
// Maintains KPI\ProdOrder\  folder files
fbMaintainFolders[10](
    NETID := '',
    PATHSTR := CONCAT(STR1 := stMetsStatus.sLocalHMIPath, STR2 := 'Modules\ME_Archive_Delete_Tool\ME_Archive_Delete_Tool.exe'),
    DIRNAME := '',
    COMNDLINE := F_CONCAT7(strString1 := cME_ARCHIVE_ACTION[2], strString2 := ' ', strString3 := CONCAT(STR1 := stMetsStatus.sBasePath, STR2 := cBASE_FOLDER_ARR[18]), strString4 := ' ', strString5 := INT_TO_STRING(stMachineConfig.nMaximumArchiveAge), strString6 := ' ', strString7 := 'FALSE'),
    START := fbMaintainDeleteTime.bOutput AND nActivateBitWord.10,
    TMOUT := cONE_SECOND); // NT_StartProcess

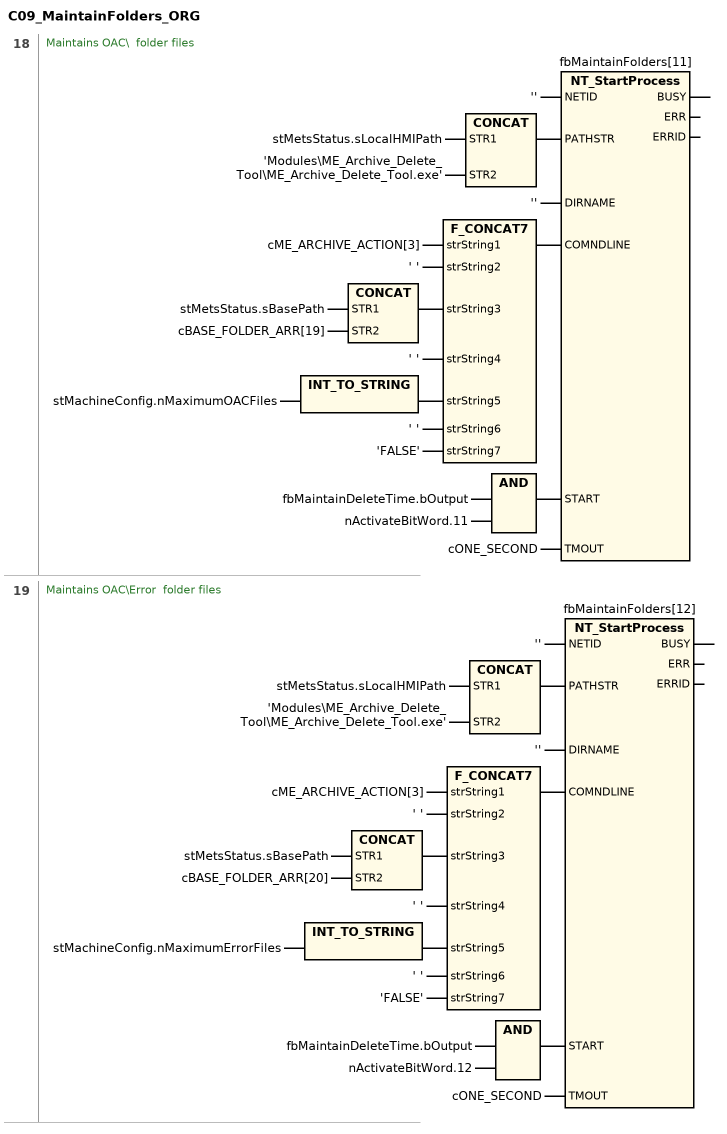
// NETWORK 18
// Maintains OAC\  folder files
fbMaintainFolders[11](
    NETID := '',
    PATHSTR := CONCAT(STR1 := stMetsStatus.sLocalHMIPath, STR2 := 'Modules\ME_Archive_Delete_Tool\ME_Archive_Delete_Tool.exe'),
    DIRNAME := '',
    COMNDLINE := F_CONCAT7(strString1 := cME_ARCHIVE_ACTION[3], strString2 := ' ', strString3 := CONCAT(STR1 := stMetsStatus.sBasePath, STR2 := cBASE_FOLDER_ARR[19]), strString4 := ' ', strString5 := INT_TO_STRING(stMachineConfig.nMaximumOACFiles), strString6 := ' ', strString7 := 'FALSE'),
    START := fbMaintainDeleteTime.bOutput AND nActivateBitWord.11,
    TMOUT := cONE_SECOND); // NT_StartProcess

// NETWORK 19
// Maintains OAC\Error  folder files
fbMaintainFolders[12](
    NETID := '',
    PATHSTR := CONCAT(STR1 := stMetsStatus.sLocalHMIPath, STR2 := 'Modules\ME_Archive_Delete_Tool\ME_Archive_Delete_Tool.exe'),
    DIRNAME := '',
    COMNDLINE := F_CONCAT7(strString1 := cME_ARCHIVE_ACTION[3], strString2 := ' ', strString3 := CONCAT(STR1 := stMetsStatus.sBasePath, STR2 := cBASE_FOLDER_ARR[20]), strString4 := ' ', strString5 := INT_TO_STRING(stMachineConfig.nMaximumErrorFiles), strString6 := ' ', strString7 := 'FALSE'),
    START := fbMaintainDeleteTime.bOutput AND nActivateBitWord.12,
    TMOUT := cONE_SECOND); // NT_StartProcess

